Omron Sysmac Studio project Meca500_V9_3_3_Omron_EthernetIP_SquareMove_Demo_V1_1 (Sysmac Studio 1.53.0.64009, StandardProject)
(* Ajouter Calculate WRF function *)

# Controller NX1P2_1040DT1: NX1P2-1040DT1 version 1.16
Task PrimaryTask (priority 4, period or condition 2000): Meca500_E001

TYPE RobotControl : STRUCT
    Deactivate : BOOL;  (* offset 0.0 *)
    Activate : BOOL;  (* offset 0.1 *)
    Home : BOOL;  (* offset 0.2 *)
    ResetError : BOOL;  (* offset 0.3 *)
    EnableSimulation : BOOL;  (* offset 0.4 *)
    EnableRecoveryMode : BOOL;  (* offset 0.5 *)
END_STRUCT END_TYPE
TYPE Meca500 : STRUCT
    Outputs : Outputs;
    Inputs : Inputs;
    CommandsID : Meca500Cmd;
END_STRUCT END_TYPE
TYPE Inputs : STRUCT
    Status : Status;  (* offset 0.0 *)
    Motion : Motion;  (* offset 4.0 *)
    Joint_Set : Joint_Set;  (* offset 16.0 *)
    EndEffector_Pose : EndEffector_Pose;  (* offset 40.0 *)
    Configurations : Configurations;  (* offset 64.0 *)
    WRF : WRF;  (* offset 68.0 *)
    TRF : TRF;  (* offset 92.0 *)
    TimeStamp : TimeStamp;  (* offset 116.0 *)
    Reserved1 : SINT;  (* offset 128.0 *)
    Reserved2 : SINT;  (* offset 132.0 *)
    Reserved3 : SINT;  (* offset 136.0 *)
    DynamicData0 : DynamicData;  (* offset 140.0 *)
    DynamicData1 : DynamicData;  (* offset 168.0 *)
    DynamicData2 : DynamicData;  (* offset 196.0 *)
    DynamicData3 : DynamicData;  (* offset 224.0 *)
END_STRUCT END_TYPE
TYPE Status : STRUCT
    Busy : BOOL;
    Activated : BOOL;
    Homed : BOOL;
    SimActivated : BOOL;
    BrakesEngaged : BOOL;
    RecoveryMode : BOOL;
    EStop : BOOL;
    Error : UINT;
END_STRUCT END_TYPE
TYPE Motion : STRUCT
    CheckPoint : UDINT;  (* offset 0.0 *)
    MoveID : UINT;  (* offset 4.0 *)
    FifoSpace : UINT;  (* offset 6.0 *)
    Paused : BOOL;  (* offset 8.0 *)
    EOB : BOOL;  (* offset 8.1 *)
    EOM : BOOL;  (* offset 8.2 *)
    FifoCleared : BOOL;  (* offset 8.3 *)
    PStop2 : BOOL;  (* offset 8.4 *)
    ExcessiveTorque : BOOL;  (* offset 8.5 *)
    PStop2Resettable : BOOL;  (* offset 8.6 *)
    OfflineProgramID : UINT;  (* offset 10.0 *)
END_STRUCT END_TYPE
TYPE Joint_Set : STRUCT
    SubIndex001 : REAL;
    SubIndex002 : REAL;
    SubIndex003 : REAL;
    SubIndex004 : REAL;
    SubIndex005 : REAL;
    SubIndex006 : REAL;
END_STRUCT END_TYPE
TYPE EndEffector_Pose : STRUCT
    SubIndex001 : REAL;
    SubIndex002 : REAL;
    SubIndex003 : REAL;
    SubIndex004 : REAL;
    SubIndex005 : REAL;
    SubIndex006 : REAL;
END_STRUCT END_TYPE
TYPE Configurations : STRUCT
    Shoulder : SINT;  (* offset 0.0 *)
    Elbow : SINT;  (* offset 1.0 *)
    Wrist : SINT;  (* offset 2.0 *)
    Turn : SINT;  (* offset 3.0 *)
END_STRUCT END_TYPE
TYPE WRF : STRUCT
    SubIndex001 : REAL;
    SubIndex002 : REAL;
    SubIndex003 : REAL;
    SubIndex004 : REAL;
    SubIndex005 : REAL;
    SubIndex006 : REAL;
END_STRUCT END_TYPE
TYPE TRF : STRUCT
    SubIndex001 : REAL;
    SubIndex002 : REAL;
    SubIndex003 : REAL;
    SubIndex004 : REAL;
    SubIndex005 : REAL;
    SubIndex006 : REAL;
END_STRUCT END_TYPE
TYPE TimeStamp : STRUCT
    Seconds : UDINT;
    MicroSeconds : UDINT;
    DynamicDataCycles : UDINT;
END_STRUCT END_TYPE
TYPE DynamicData : STRUCT
    DynamicDataType : UDINT;
    DynamicDataValue0 : REAL;
    DynamicDataValue1 : REAL;
    DynamicDataValue2 : REAL;
    DynamicDataValue3 : REAL;
    DynamicDataValue4 : REAL;
    DynamicDataValue5 : REAL;
END_STRUCT END_TYPE
TYPE Outputs : STRUCT
    RobotControl : RobotControl;  (* offset 0.0 *)
    MotionControl : MotionControl;  (* offset 4.0 *)
    MotionCommand : MotionCommand;  (* offset 8.0 *)
    HostTime : UDINT;  (* offset 36.0 *)
    BrakesControlAllowed : BOOL;  (* offset 40.0 *)
    BrakesEngaged : BOOL;  (* offset 40.1 *)
    DynamicDataCfg0 : UDINT;  (* offset 44.0 *)
    DynamicDataCfg1 : UDINT;  (* offset 48.0 *)
    DynamicDataCfg2 : UDINT;  (* offset 52.0 *)
    DynamicDataCfg3 : UDINT;  (* offset 56.0 *)
END_STRUCT END_TYPE
TYPE MotionControl : STRUCT
    MoveID : UINT;  (* offset 0.0 *)
    Setpoint : BOOL;  (* offset 2.0 *)
    Pause : BOOL;  (* offset 2.1 *)
    CleaMove : BOOL;  (* offset 2.2 *)
    ResetPStop2 : BOOL;  (* offset 2.3 *)
END_STRUCT END_TYPE
TYPE MotionCommand : STRUCT
    MoveCommand : UDINT;  (* offset 0.0 *)
    MoveSubIndex001 : REAL;  (* offset 4.0 *)
    MoveSubIndex002 : REAL;  (* offset 8.0 *)
    MoveSubIndex003 : REAL;  (* offset 12.0 *)
    MoveSubIndex004 : REAL;  (* offset 16.0 *)
    MoveSubIndex005 : REAL;  (* offset 20.0 *)
    MoveSubIndex006 : REAL;  (* offset 24.0 *)
END_STRUCT END_TYPE
TYPE Meca500Cmd : (NoCmd := 0, MoveJoints := 1, MovePose := 2, MoveLin := 3, MoveLinRelTrf := 4, MoveLinRelWrf := 5, Delay := 6, SetBlending := 7, SetJointVel := 8, SetJointAcc := 9, SetCartAngVel := 10, SetCartLinVel := 11, SetCartAcc := 12, SetTrf := 13, SetWrf := 14, SetConf := 15, SetAutoConf := 16, SetCheckpoint := 17, Gripper := 18, SetGripperVel := 19, SetGripperForce := 20, MoveJointsVel := 21, MoveLinVelWrf := 22, MoveLinVelTrf := 23, SetVelTimeout := 24, SetConfTurn := 25, SetAutoConfTurn := 26, SetTorqueLimits := 27, SetTorquesLimitCfg := 28, MoveJointsRel := 29, SetValveState := 30, SetGripperRange := 31, MoveGripper := 32, SetJointVelLimit := 33, StartProgram := 100); END_TYPE

VAR_GLOBAL
    E001 : Meca500;  (* Robot Structure *)
    E001_Inputs : Inputs;  (* EthernetIp Inputs; network input *)
    E001_Outputs : Outputs;  (* EthernetIP Outputs; network output *)
END_VAR
VAR_GLOBAL CONSTANT
    Pi : REAL := 3.141592653589793238;
END_VAR

PROGRAM Meca500_E001
VAR
    Activate : BOOL;
    Deactivate : BOOL;
    Home : BOOL;
    ResetError : BOOL;
    Pause : BOOL;
    RecoveryMode : BOOL;
    StepSquareMove : INT;
    StartSequence : BOOL;
    SequenceActive : BOOL;
    SetCheckpoint1Buffered : BOOL;
    SetCartLinVel1Buffered : BOOL;
    MoveJoint1Buffered : BOOL;
    MovePose1Buffered : BOOL;
    MoveLin1Buffered : BOOL;
    Argument : ARRAY[0..5] OF real;
    SetCheckpoint1 : Meca500_SetCheckpoint;
    SetCartLinVel1 : Meca500_SetCartLinVel;
    MoveJoints1 : Meca500_MoveJoints;
    MovePose1 : Meca500_MovePose;
    MoveLin1 : Meca500_MoveLin;
END_VAR
VAR_EXTERNAL
    E001 : Meca500;
    E001_Inputs : Inputs;
    E001_Outputs : Outputs;
END_VAR
VAR
    _e1 : R_TRIG;
END_VAR

(* Section IOs: ladder, written here as Structured Text *)

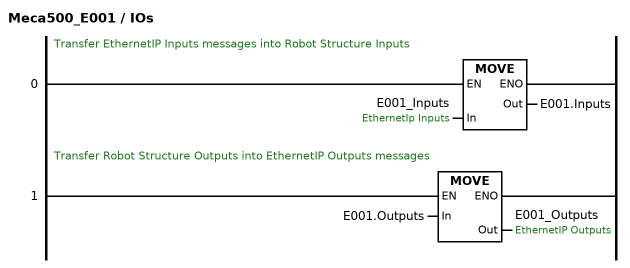
(* Rung 0: Transfer EthernetIP Inputs messages into Robot Structure Inputs *)
E001.Inputs := E001_Inputs;
(* Rung 1: Transfer Robot Structure Outputs into EthernetIP Outputs messages *)
E001_Outputs := E001.Outputs;

(* Section Robot_Control: ladder, written here as Structured Text *)

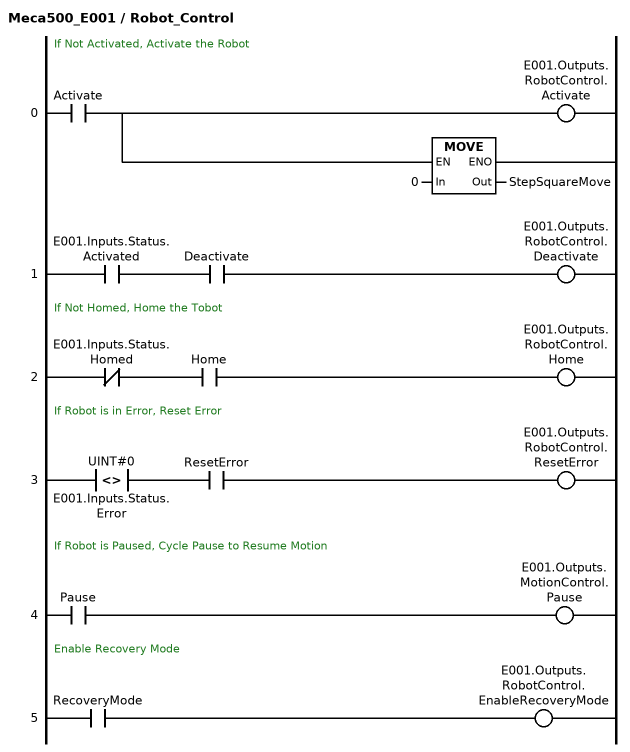
(* Rung 0: If Not Activated, Activate the Robot *)
E001.Outputs.RobotControl.Activate := Activate;
IF Activate THEN StepSquareMove := 0; END_IF;
(* Rung 1 *)
E001.Outputs.RobotControl.Deactivate := E001.Inputs.Status.Activated AND Deactivate;
(* Rung 2: If Not Homed, Home the Tobot *)
E001.Outputs.RobotControl.Home := NOT E001.Inputs.Status.Homed AND Home;
(* Rung 3: If Robot is in Error, Reset Error *)
E001.Outputs.RobotControl.ResetError := (UINT#0 <> E001.Inputs.Status.Error) AND ResetError;
(* Rung 4: If Robot is Paused, Cycle Pause to Resume Motion *)
E001.Outputs.MotionControl.Pause := Pause;
(* Rung 5: Enable Recovery Mode *)
E001.Outputs.RobotControl.EnableRecoveryMode := RecoveryMode;

(* Section Sequence: ladder, written here as Structured Text *)

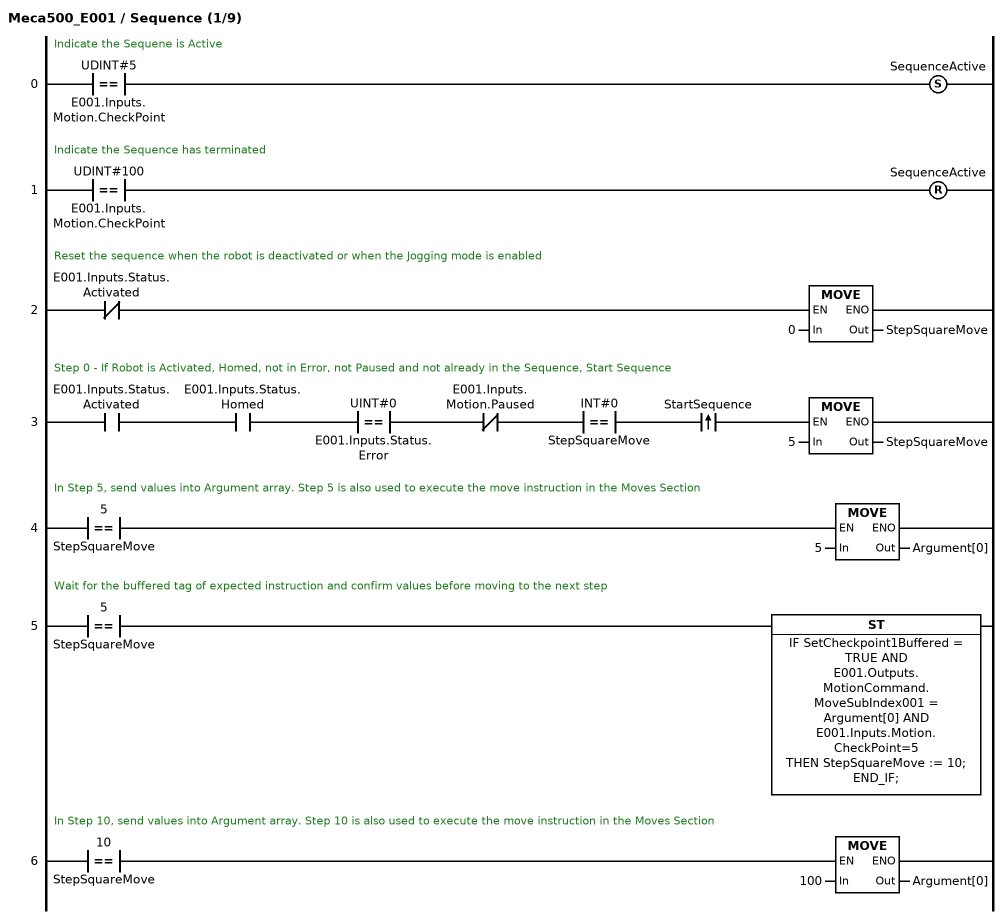
(* Rung 0: Indicate the Sequene is Active *)
IF UDINT#5 = E001.Inputs.Motion.CheckPoint THEN SequenceActive := TRUE; END_IF;
(* Rung 1: Indicate the Sequence has terminated *)
IF UDINT#100 = E001.Inputs.Motion.CheckPoint THEN SequenceActive := FALSE; END_IF;
(* Rung 2: Reset the sequence when the robot is deactivated or when the Jogging mode is enabled *)
IF NOT E001.Inputs.Status.Activated THEN StepSquareMove := 0; END_IF;
(* Rung 3: Step 0 - If Robot is Activated, Homed, not in Error, not Paused and not already in the Sequence, Start Sequence *)
_e1(CLK := StartSequence);
IF E001.Inputs.Status.Activated AND E001.Inputs.Status.Homed AND (UINT#0 = E001.Inputs.Status.Error) AND NOT E001.Inputs.Motion.Paused AND (INT#0 = StepSquareMove) AND _e1.Q THEN
    StepSquareMove := 5;
END_IF;
(* Rung 4: In Step 5, send values into Argument array. Step 5 is also used to execute the move instruction in the Moves Section *)
IF 5 = StepSquareMove THEN Argument[0] := 5; END_IF;
(* Rung 5: Wait for the buffered tag of expected instruction and confirm values before moving to the next step *)
IF 5 = StepSquareMove THEN
    IF SetCheckpoint1Buffered = TRUE AND
    	E001.Outputs.MotionCommand.MoveSubIndex001 = Argument[0] AND
    	E001.Inputs.Motion.CheckPoint=5
    	THEN StepSquareMove := 10;
    END_IF;
END_IF;
(* Rung 6: In Step 10, send values into Argument array. Step 10 is also used to execute the move instruction in the Moves Section *)
IF 10 = StepSquareMove THEN Argument[0] := 100; END_IF;

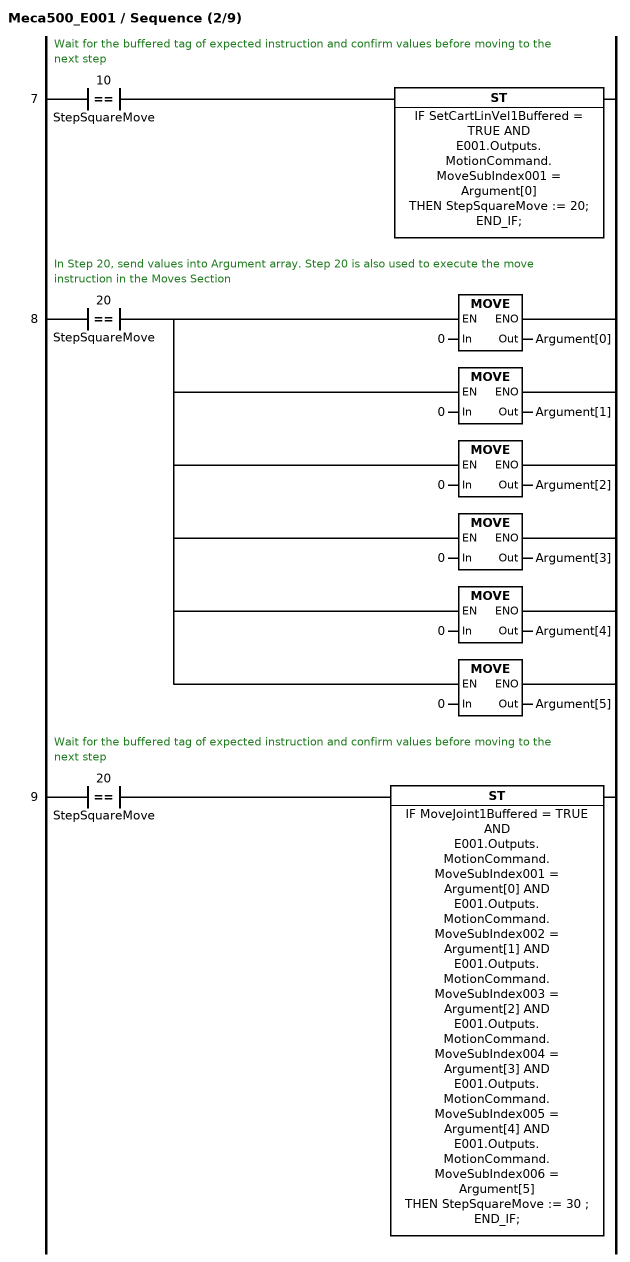
(* Rung 7: Wait for the buffered tag of expected instruction and confirm values before moving to the next step *)
IF 10 = StepSquareMove THEN
    IF SetCartLinVel1Buffered = TRUE AND
    	E001.Outputs.MotionCommand.MoveSubIndex001 = Argument[0]
    	THEN StepSquareMove := 20;
    END_IF;
END_IF;
(* Rung 8: In Step 20, send values into Argument array. Step 20 is also used to execute the move instruction in the Moves Section *)
IF 20 = StepSquareMove THEN
    Argument[0] := 0;
    Argument[1] := 0;
    Argument[2] := 0;
    Argument[3] := 0;
    Argument[4] := 0;
    Argument[5] := 0;
END_IF;
(* Rung 9: Wait for the buffered tag of expected instruction and confirm values before moving to the next step *)
IF 20 = StepSquareMove THEN
    IF MoveJoint1Buffered = TRUE AND
    	E001.Outputs.MotionCommand.MoveSubIndex001 = Argument[0] AND
    	E001.Outputs.MotionCommand.MoveSubIndex002 = Argument[1] AND
    	E001.Outputs.MotionCommand.MoveSubIndex003 = Argument[2] AND
    	E001.Outputs.MotionCommand.MoveSubIndex004 = Argument[3] AND
    	E001.Outputs.MotionCommand.MoveSubIndex005 = Argument[4] AND
    	E001.Outputs.MotionCommand.MoveSubIndex006 = Argument[5] 
    	THEN StepSquareMove := 30 ;
    END_IF;
END_IF;

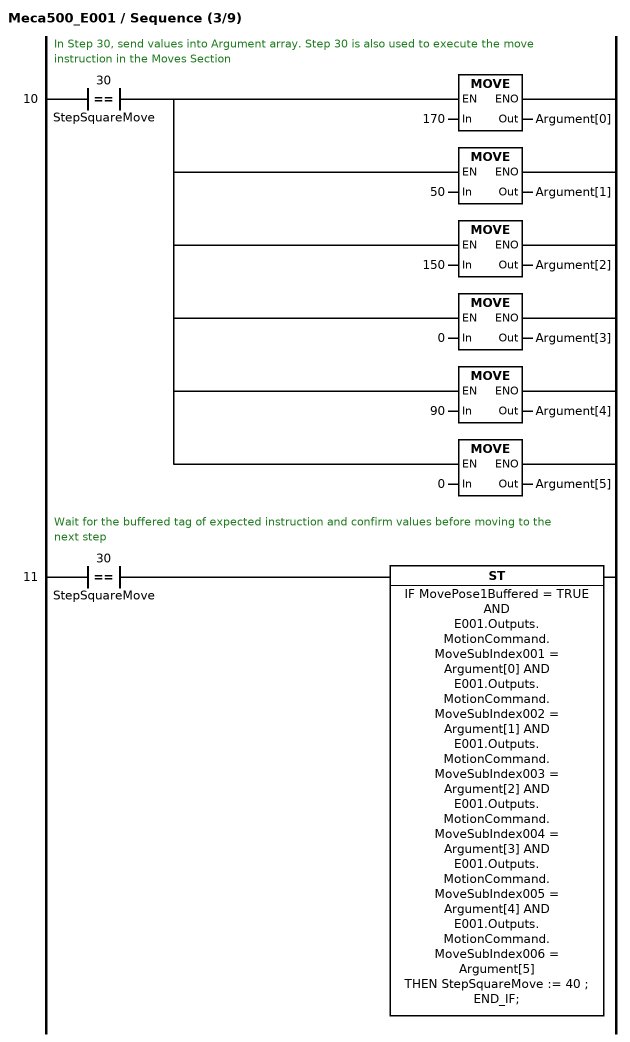
(* Rung 10: In Step 30, send values into Argument array. Step 30 is also used to execute the move instruction in the Moves Section *)
IF 30 = StepSquareMove THEN
    Argument[0] := 170;
    Argument[1] := 50;
    Argument[2] := 150;
    Argument[3] := 0;
    Argument[4] := 90;
    Argument[5] := 0;
END_IF;
(* Rung 11: Wait for the buffered tag of expected instruction and confirm values before moving to the next step *)
IF 30 = StepSquareMove THEN
    IF MovePose1Buffered = TRUE AND
    	E001.Outputs.MotionCommand.MoveSubIndex001 = Argument[0] AND
    	E001.Outputs.MotionCommand.MoveSubIndex002 = Argument[1] AND
    	E001.Outputs.MotionCommand.MoveSubIndex003 = Argument[2] AND
    	E001.Outputs.MotionCommand.MoveSubIndex004 = Argument[3] AND
    	E001.Outputs.MotionCommand.MoveSubIndex005 = Argument[4] AND
    	E001.Outputs.MotionCommand.MoveSubIndex006 = Argument[5] 
    	THEN StepSquareMove := 40 ;
    END_IF;
END_IF;

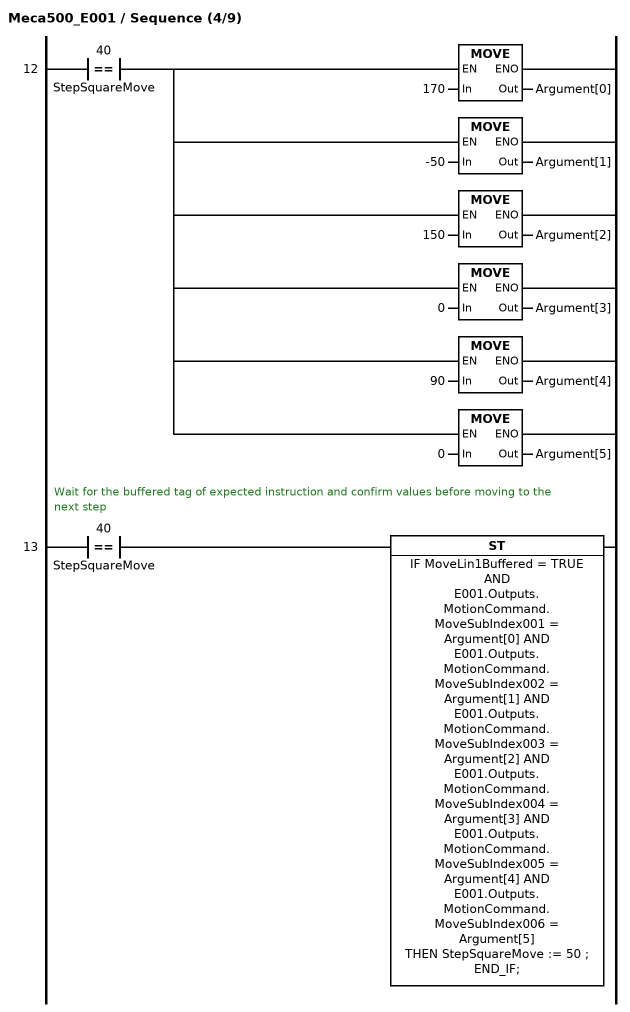
(* Rung 12 *)
IF 40 = StepSquareMove THEN
    Argument[0] := 170;
    Argument[1] := -50;
    Argument[2] := 150;
    Argument[3] := 0;
    Argument[4] := 90;
    Argument[5] := 0;
END_IF;
(* Rung 13: Wait for the buffered tag of expected instruction and confirm values before moving to the next step *)
IF 40 = StepSquareMove THEN
    IF MoveLin1Buffered = TRUE AND
    	E001.Outputs.MotionCommand.MoveSubIndex001 = Argument[0] AND
    	E001.Outputs.MotionCommand.MoveSubIndex002 = Argument[1] AND
    	E001.Outputs.MotionCommand.MoveSubIndex003 = Argument[2] AND
    	E001.Outputs.MotionCommand.MoveSubIndex004 = Argument[3] AND
    	E001.Outputs.MotionCommand.MoveSubIndex005 = Argument[4] AND
    	E001.Outputs.MotionCommand.MoveSubIndex006 = Argument[5] 
    	THEN StepSquareMove := 50 ;
    END_IF;
END_IF;

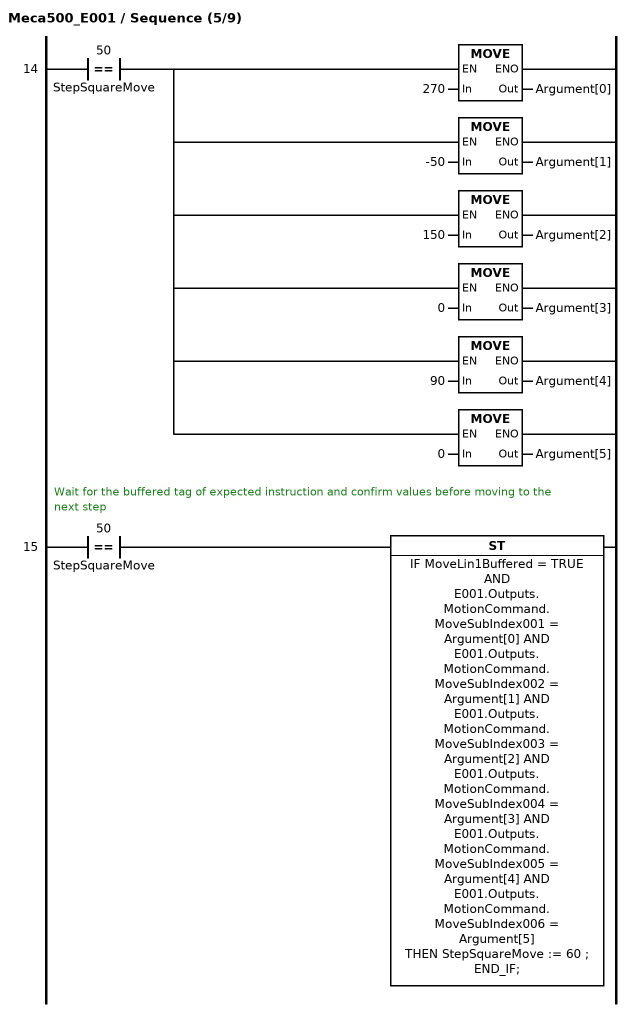
(* Rung 14 *)
IF 50 = StepSquareMove THEN
    Argument[0] := 270;
    Argument[1] := -50;
    Argument[2] := 150;
    Argument[3] := 0;
    Argument[4] := 90;
    Argument[5] := 0;
END_IF;
(* Rung 15: Wait for the buffered tag of expected instruction and confirm values before moving to the next step *)
IF 50 = StepSquareMove THEN
    IF MoveLin1Buffered = TRUE AND
    	E001.Outputs.MotionCommand.MoveSubIndex001 = Argument[0] AND
    	E001.Outputs.MotionCommand.MoveSubIndex002 = Argument[1] AND
    	E001.Outputs.MotionCommand.MoveSubIndex003 = Argument[2] AND
    	E001.Outputs.MotionCommand.MoveSubIndex004 = Argument[3] AND
    	E001.Outputs.MotionCommand.MoveSubIndex005 = Argument[4] AND
    	E001.Outputs.MotionCommand.MoveSubIndex006 = Argument[5] 
    	THEN StepSquareMove := 60 ;
    END_IF;
END_IF;

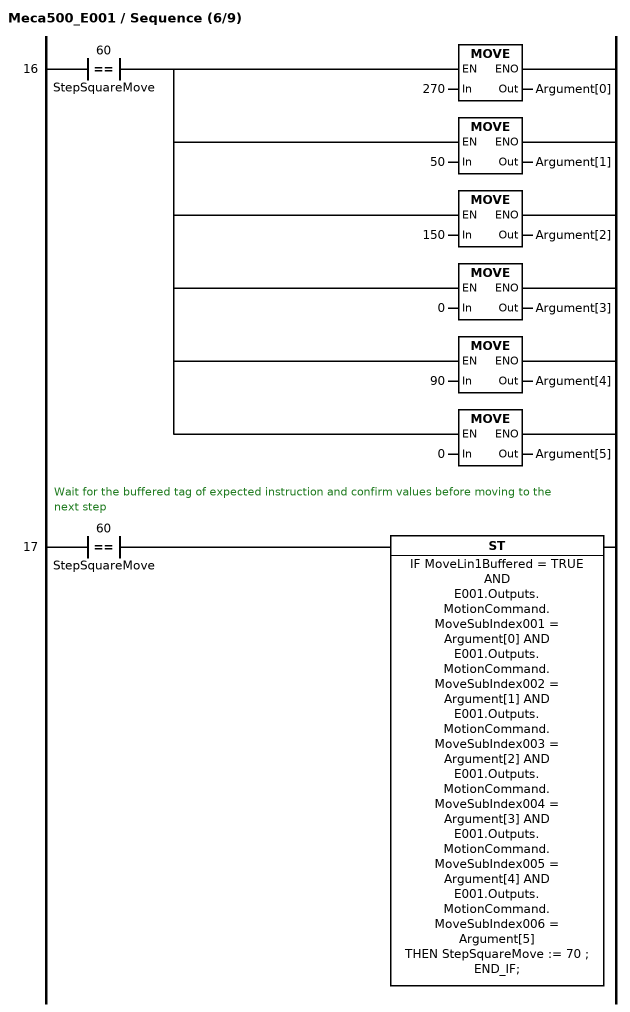
(* Rung 16 *)
IF 60 = StepSquareMove THEN
    Argument[0] := 270;
    Argument[1] := 50;
    Argument[2] := 150;
    Argument[3] := 0;
    Argument[4] := 90;
    Argument[5] := 0;
END_IF;
(* Rung 17: Wait for the buffered tag of expected instruction and confirm values before moving to the next step *)
IF 60 = StepSquareMove THEN
    IF MoveLin1Buffered = TRUE AND
    	E001.Outputs.MotionCommand.MoveSubIndex001 = Argument[0] AND
    	E001.Outputs.MotionCommand.MoveSubIndex002 = Argument[1] AND
    	E001.Outputs.MotionCommand.MoveSubIndex003 = Argument[2] AND
    	E001.Outputs.MotionCommand.MoveSubIndex004 = Argument[3] AND
    	E001.Outputs.MotionCommand.MoveSubIndex005 = Argument[4] AND
    	E001.Outputs.MotionCommand.MoveSubIndex006 = Argument[5] 
    	THEN StepSquareMove := 70 ;
    END_IF;
END_IF;

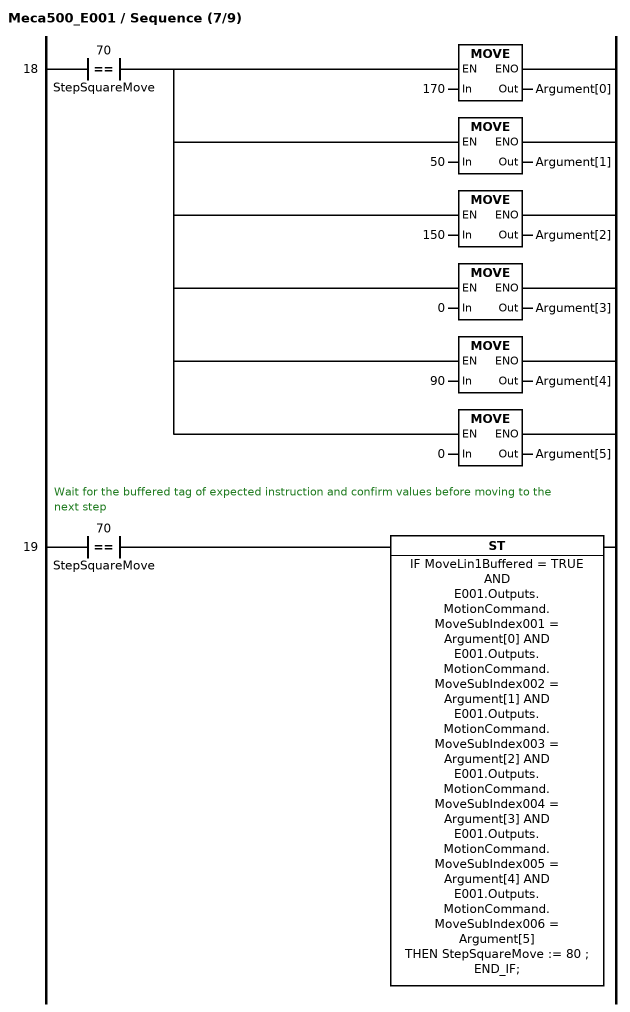
(* Rung 18 *)
IF 70 = StepSquareMove THEN
    Argument[0] := 170;
    Argument[1] := 50;
    Argument[2] := 150;
    Argument[3] := 0;
    Argument[4] := 90;
    Argument[5] := 0;
END_IF;
(* Rung 19: Wait for the buffered tag of expected instruction and confirm values before moving to the next step *)
IF 70 = StepSquareMove THEN
    IF MoveLin1Buffered = TRUE AND
    	E001.Outputs.MotionCommand.MoveSubIndex001 = Argument[0] AND
    	E001.Outputs.MotionCommand.MoveSubIndex002 = Argument[1] AND
    	E001.Outputs.MotionCommand.MoveSubIndex003 = Argument[2] AND
    	E001.Outputs.MotionCommand.MoveSubIndex004 = Argument[3] AND
    	E001.Outputs.MotionCommand.MoveSubIndex005 = Argument[4] AND
    	E001.Outputs.MotionCommand.MoveSubIndex006 = Argument[5] 
    	THEN StepSquareMove := 80 ;
    END_IF;
END_IF;

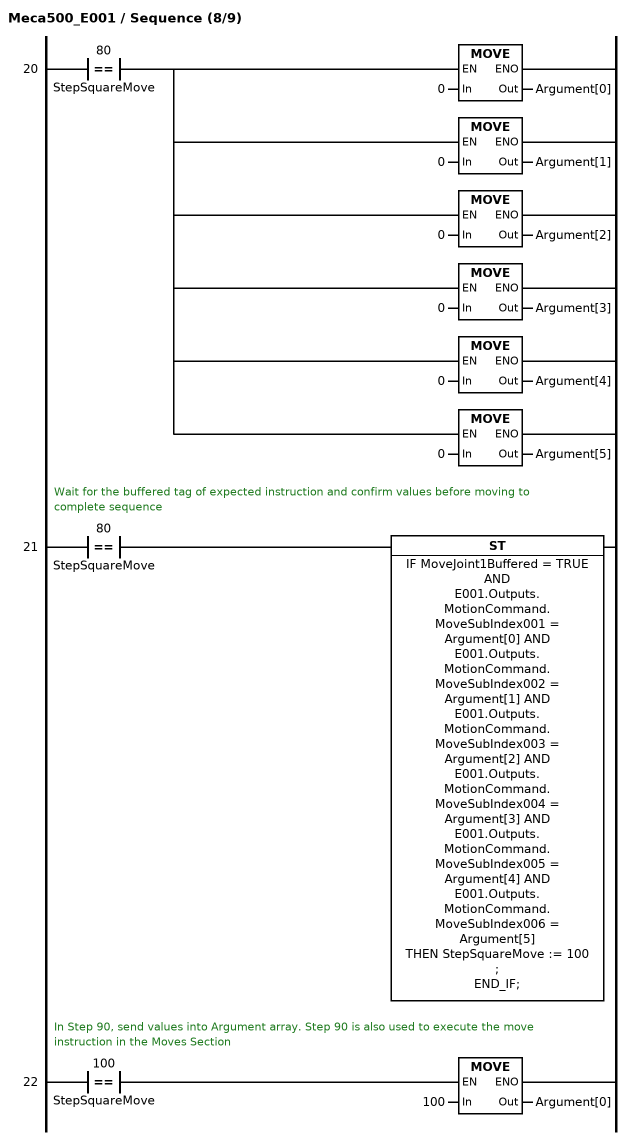
(* Rung 20 *)
IF 80 = StepSquareMove THEN
    Argument[0] := 0;
    Argument[1] := 0;
    Argument[2] := 0;
    Argument[3] := 0;
    Argument[4] := 0;
    Argument[5] := 0;
END_IF;
(* Rung 21: Wait for the buffered tag of expected instruction and confirm values before moving to complete sequence *)
IF 80 = StepSquareMove THEN
    IF MoveJoint1Buffered = TRUE AND
    	E001.Outputs.MotionCommand.MoveSubIndex001 = Argument[0] AND
    	E001.Outputs.MotionCommand.MoveSubIndex002 = Argument[1] AND
    	E001.Outputs.MotionCommand.MoveSubIndex003 = Argument[2] AND
    	E001.Outputs.MotionCommand.MoveSubIndex004 = Argument[3] AND
    	E001.Outputs.MotionCommand.MoveSubIndex005 = Argument[4] AND
    	E001.Outputs.MotionCommand.MoveSubIndex006 = Argument[5] 
    	THEN StepSquareMove := 100 ;
    END_IF;
END_IF;
(* Rung 22: In Step 90, send values into Argument array. Step 90 is also used to execute the move instruction in the Moves Section *)
IF 100 = StepSquareMove THEN Argument[0] := 100; END_IF;

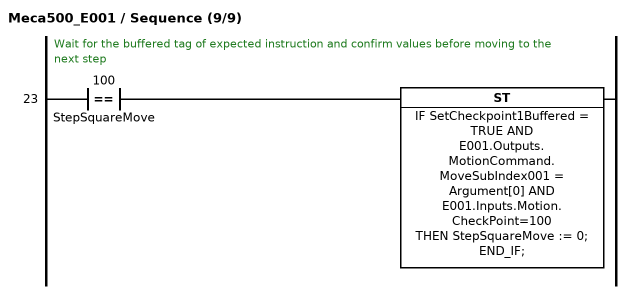
(* Rung 23: Wait for the buffered tag of expected instruction and confirm values before moving to the next step *)
IF 100 = StepSquareMove THEN
    IF SetCheckpoint1Buffered = TRUE AND
    	E001.Outputs.MotionCommand.MoveSubIndex001 = Argument[0] AND
    	E001.Inputs.Motion.CheckPoint=100
    	THEN StepSquareMove := 0;
    END_IF;
END_IF;

(* Section Instructions: ladder, written here as Structured Text *)

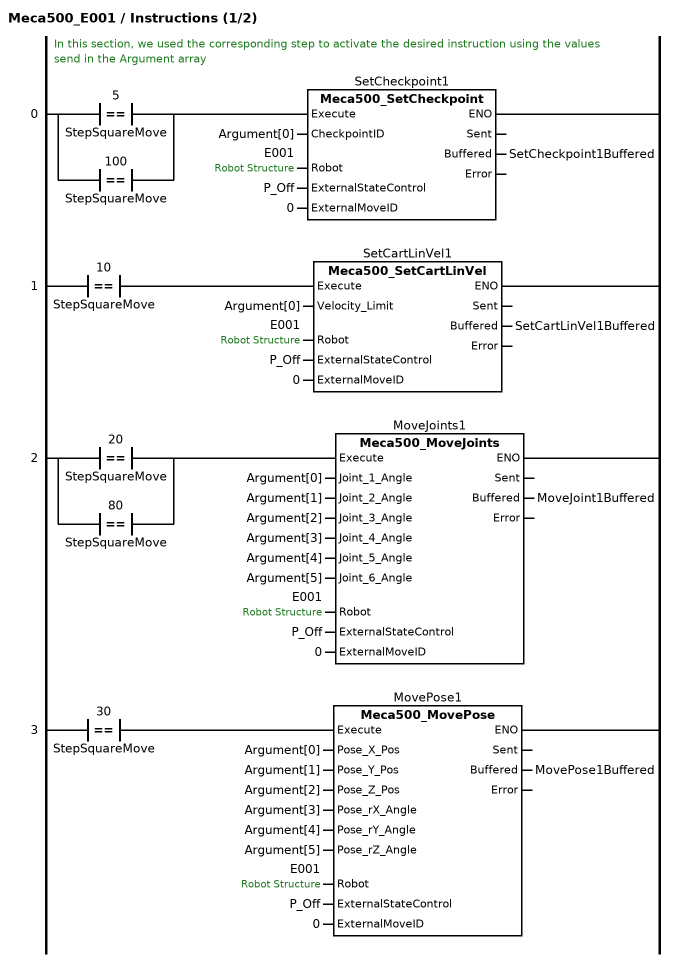
(* Rung 0: In this section, we used the corresponding step to activate the desired instruction using the values send in the Argument array *)
SetCheckpoint1(Execute := (5 = StepSquareMove) OR (100 = StepSquareMove), CheckpointID := Argument[0], Robot := E001, ExternalStateControl := P_Off, ExternalMoveID := 0, Buffered => SetCheckpoint1Buffered);
(* Rung 1 *)
SetCartLinVel1(Execute := 10 = StepSquareMove, Velocity_Limit := Argument[0], Robot := E001, ExternalStateControl := P_Off, ExternalMoveID := 0, Buffered => SetCartLinVel1Buffered);
(* Rung 2 *)
MoveJoints1(Execute := (20 = StepSquareMove) OR (80 = StepSquareMove), Joint_1_Angle := Argument[0], Joint_2_Angle := Argument[1], Joint_3_Angle := Argument[2], Joint_4_Angle := Argument[3], Joint_5_Angle := Argument[4], Joint_6_Angle := Argument[5], Robot := E001, ExternalStateControl := P_Off, ExternalMoveID := 0, Buffered => MoveJoint1Buffered);
(* Rung 3 *)
MovePose1(Execute := 30 = StepSquareMove, Pose_X_Pos := Argument[0], Pose_Y_Pos := Argument[1], Pose_Z_Pos := Argument[2], Pose_rX_Angle := Argument[3], Pose_rY_Angle := Argument[4], Pose_rZ_Angle := Argument[5], Robot := E001, ExternalStateControl := P_Off, ExternalMoveID := 0, Buffered => MovePose1Buffered);

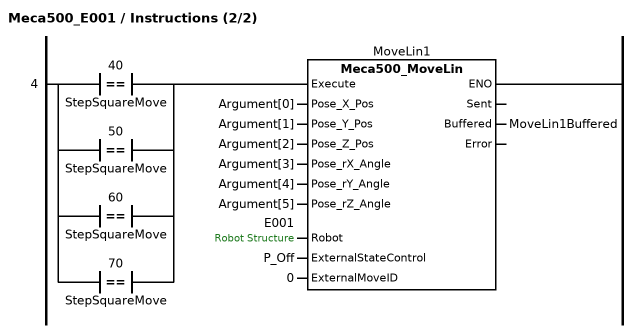
(* Rung 4 *)
MoveLin1(Execute := (40 = StepSquareMove) OR (50 = StepSquareMove) OR (60 = StepSquareMove) OR (70 = StepSquareMove), Pose_X_Pos := Argument[0], Pose_Y_Pos := Argument[1], Pose_Z_Pos := Argument[2], Pose_rX_Angle := Argument[3], Pose_rY_Angle := Argument[4], Pose_rZ_Angle := Argument[5], Robot := E001, ExternalStateControl := P_Off, ExternalMoveID := 0, Buffered => MoveLin1Buffered);
END_PROGRAM

FUNCTION atan2 : lREAL
VAR_INPUT
    y : lREAL;
    x : lREAL;
END_VAR
VAR_EXTERNAL CONSTANT
    Pi : REAL;
END_VAR
IF x > 0 THEN
	Atan2:=ATAN(y/x);
ELSIF x<0 AND y>=0 THEN
	Atan2:=ATAN(y/x)+Pi;
ELSIF  x<0 AND y<0 THEN
	Atan2:=ATAN(y/x)-Pi;
ELSIF  x=0 AND y>0 THEN
	Atan2:=Pi/2;
ELSIF  x=0 AND y<0 THEN
	Atan2:=-Pi/2;
END_IF;
END_FUNCTION

FUNCTION_BLOCK Meca500_Delay
VAR
    Output_Params : array[1..6] of real;
    FirstScan : BOOL := False;
END_VAR
VAR_INPUT
    Execute : BOOL;
    Seconds : REAL;
END_VAR
VAR_OUTPUT
    Sent : BOOL;
    Buffered : BOOL;
    Error : BOOL;
END_VAR
VAR_IN_OUT
    Robot : Meca500;
END_VAR
VAR_INPUT
    ExternalStateControl : BOOL;
    ExternalMoveID : UINT;
END_VAR
IF Execute THEN	
	(*Collect Inputs and store them locally*)
	Output_Params[1]:=Seconds;
	Output_Params[2]:=0;
	Output_Params[3]:=0;
	Output_Params[4]:=0;
	Output_Params[5]:=0;
	Output_Params[6]:=0;


	(* If Values have change, Reinitialise Outputs*)

	IF FirstScan=0 OR 
		Robot.Outputs.MotionCommand.MoveSubIndex001 <> Output_Params[1] OR 
		Robot.Outputs.MotionCommand.MoveSubIndex002 <> Output_Params[2] OR 
		Robot.Outputs.MotionCommand.MoveSubIndex003 <> Output_Params[3] OR
		Robot.Outputs.MotionCommand.MoveSubIndex004 <> Output_Params[4] OR 
		Robot.Outputs.MotionCommand.MoveSubIndex005 <> Output_Params[5] OR 
		Robot.Outputs.MotionCommand.MoveSubIndex006 <> Output_Params[6] 
	THEN
		Buffered := FALSE;
		Sent := FALSE;
	END_IF;


	(*if not in legacy mode, Act Setpoint*)
	IF Robot.Outputs.MotionControl.MoveID <> 0 THEN
	    Robot.Outputs.MotionControl.SetPoint := TRUE;
	END_IF;

	(* To send _Move, send _Move ID *)
	IF NOT Buffered AND NOT Sent THEN
	    
	    Robot.Outputs.MotionCommand.MoveCommand	:= EnumToNum(Meca500Cmd#Delay);
	    Robot.Outputs.MotionCommand.MoveSubIndex001 := Output_Params[1];
		Robot.Outputs.MotionCommand.MoveSubIndex002 := Output_Params[2];
		Robot.Outputs.MotionCommand.MoveSubIndex003 := Output_Params[3];
		Robot.Outputs.MotionCommand.MoveSubIndex004 := Output_Params[4];
		Robot.Outputs.MotionCommand.MoveSubIndex005 := Output_Params[5];
		Robot.Outputs.MotionCommand.MoveSubIndex006 := Output_Params[6];
	    
	    IF ExternalStateControl THEN
	        IF ExternalMoveID <> 0 AND ExternalMoveID <> 32060 AND ExternalMoveID <> 32061 THEN
	            Robot.Outputs.MotionControl.MoveID := ExternalMoveID;
	            Sent := TRUE;
	        END_IF;
	        
	    ELSE (*Not External Control*)
	        IF Robot.Outputs.MotionControl.MoveID = 32060 THEN
	            Robot.Outputs.MotionControl.MoveID := 32061;
	        ELSIF Robot.Outputs.MotionControl.MoveID = 32061 THEN
	            Robot.Outputs.MotionControl.MoveID := 32060;
	        ELSIF Robot.Outputs.MotionControl.MoveID <> 32060 OR Robot.Outputs.MotionControl.MoveID <> 32061 THEN
	            Robot.Outputs.MotionControl.MoveID := 32060;
	        END_IF;
	        Sent := TRUE;
	    END_IF;
	END_IF;

	(* Check if command has been sent, if so, check if it was received *)
	IF Sent AND
	    Robot.Outputs.MotionCommand.MoveCommand = EnumToNum(Meca500Cmd#Delay) AND
	    Robot.Outputs.MotionCommand.MoveSubIndex001 = Output_Params[1] AND 
		Robot.Outputs.MotionCommand.MoveSubIndex002 = Output_Params[2] AND 
		Robot.Outputs.MotionCommand.MoveSubIndex003 = Output_Params[3] AND 
		Robot.Outputs.MotionCommand.MoveSubIndex004 = Output_Params[4] AND 
		Robot.Outputs.MotionCommand.MoveSubIndex005 = Output_Params[5] AND 
		Robot.Outputs.MotionCommand.MoveSubIndex006 = Output_Params[6] AND
		Robot.Inputs.Motion.MoveID = Robot.Outputs.MotionControl.MoveID 
	THEN
		 Buffered := TRUE;
	END_IF;


	(*If External _Move ID is equal to Internal, raise an error*)
	IF ExternalMoveID = 32060 OR ExternalMoveID = 32061 THEN
	    Error := TRUE;
	END_IF;

	FirstScan := TRUE;
ELSE
	FirstScan := False;
	Sent := FALSE;
	Buffered := FALSE;
END_IF;
END_FUNCTION_BLOCK

FUNCTION_BLOCK Meca500_Gripper
VAR
    Output_Params : array[1..6] of real;
    FirstScan : BOOL := False;
END_VAR
VAR_INPUT
    Execute : BOOL;
    Open : REAL;
END_VAR
VAR_OUTPUT
    Sent : BOOL;
    Buffered : BOOL;
    Error : BOOL;
END_VAR
VAR_IN_OUT
    Robot : Meca500;
END_VAR
VAR_INPUT
    ExternalStateControl : BOOL;
    ExternalMoveID : UINT;
END_VAR
IF Execute THEN	
	(*Collect Inputs and store them locally*)
	Output_Params[1]:=Open;
	Output_Params[2]:=0;
	Output_Params[3]:=0;
	Output_Params[4]:=0;
	Output_Params[5]:=0;
	Output_Params[6]:=0;


	(* If Values have change, Reinitialise Outputs*)

	IF FirstScan=0 OR 
		Robot.Outputs.MotionCommand.MoveSubIndex001 <> Output_Params[1] OR 
		Robot.Outputs.MotionCommand.MoveSubIndex002 <> Output_Params[2] OR 
		Robot.Outputs.MotionCommand.MoveSubIndex003 <> Output_Params[3] OR
		Robot.Outputs.MotionCommand.MoveSubIndex004 <> Output_Params[4] OR 
		Robot.Outputs.MotionCommand.MoveSubIndex005 <> Output_Params[5] OR 
		Robot.Outputs.MotionCommand.MoveSubIndex006 <> Output_Params[6] 
	THEN
		Buffered := FALSE;
		Sent := FALSE;
	END_IF;


	(*if not in legacy mode, Act Setpoint*)
	IF Robot.Outputs.MotionControl.MoveID <> 0 THEN
	    Robot.Outputs.MotionControl.SetPoint := TRUE;
	END_IF;

	(* To send _Move, send _Move ID *)
	IF NOT Buffered AND NOT Sent THEN
	    
	    Robot.Outputs.MotionCommand.MoveCommand	:= EnumToNum(Meca500Cmd#Gripper);
	    Robot.Outputs.MotionCommand.MoveSubIndex001 := Output_Params[1];
		Robot.Outputs.MotionCommand.MoveSubIndex002 := Output_Params[2];
		Robot.Outputs.MotionCommand.MoveSubIndex003 := Output_Params[3];
		Robot.Outputs.MotionCommand.MoveSubIndex004 := Output_Params[4];
		Robot.Outputs.MotionCommand.MoveSubIndex005 := Output_Params[5];
		Robot.Outputs.MotionCommand.MoveSubIndex006 := Output_Params[6];
	    
	    IF ExternalStateControl THEN
	        IF ExternalMoveID <> 0 AND ExternalMoveID <> 32180 AND ExternalMoveID <> 32181 THEN
	            Robot.Outputs.MotionControl.MoveID := ExternalMoveID;
	            Sent := TRUE;
	        END_IF;
	        
	    ELSE (*Not External Control*)
	        IF Robot.Outputs.MotionControl.MoveID = 32180 THEN
	            Robot.Outputs.MotionControl.MoveID := 32181;
	        ELSIF Robot.Outputs.MotionControl.MoveID = 32181 THEN
	            Robot.Outputs.MotionControl.MoveID := 32180;
	        ELSIF Robot.Outputs.MotionControl.MoveID <> 32180 OR Robot.Outputs.MotionControl.MoveID <> 32181 THEN
	            Robot.Outputs.MotionControl.MoveID := 32180;
	        END_IF;
	        Sent := TRUE;
	    END_IF;
	END_IF;

	(* Check if command has been sent, if so, check if it was received *)
	IF Sent AND
	    Robot.Outputs.MotionCommand.MoveCommand = EnumToNum(Meca500Cmd#Gripper) AND
	    Robot.Outputs.MotionCommand.MoveSubIndex001 = Output_Params[1] AND 
		Robot.Outputs.MotionCommand.MoveSubIndex002 = Output_Params[2] AND 
		Robot.Outputs.MotionCommand.MoveSubIndex003 = Output_Params[3] AND 
		Robot.Outputs.MotionCommand.MoveSubIndex004 = Output_Params[4] AND 
		Robot.Outputs.MotionCommand.MoveSubIndex005 = Output_Params[5] AND 
		Robot.Outputs.MotionCommand.MoveSubIndex006 = Output_Params[6] AND
		Robot.Inputs.Motion.MoveID = Robot.Outputs.MotionControl.MoveID 
	THEN
		 Buffered := TRUE;
	END_IF;


	(*If External _Move ID is equal to Internal, raise an error*)
	IF ExternalMoveID = 32180 OR ExternalMoveID = 32181 THEN
	    Error := TRUE;
	END_IF;

	FirstScan := TRUE;
ELSE
	FirstScan := False;
	Sent := FALSE;
	Buffered := FALSE;
END_IF;
END_FUNCTION_BLOCK

FUNCTION_BLOCK Meca500_MoveGripper
VAR
    Output_Params : array[1..6] of real;
    FirstScan : BOOL := False;
END_VAR
VAR_INPUT
    Execute : BOOL;
    mm : REAL;
END_VAR
VAR_OUTPUT
    Sent : BOOL;
    Buffered : BOOL;
    Error : BOOL;
END_VAR
VAR_IN_OUT
    Robot : Meca500;
END_VAR
VAR_INPUT
    ExternalStateControl : BOOL;
    ExternalMoveID : UINT;
END_VAR
IF Execute THEN	
	(*Collect Inputs and store them locally*)
	Output_Params[1]:=mm;
	Output_Params[2]:=0;
	Output_Params[3]:=0;
	Output_Params[4]:=0;
	Output_Params[5]:=0;
	Output_Params[6]:=0;


	(* If Values have change, Reinitialise Outputs*)

	IF FirstScan=0 OR 
		Robot.Outputs.MotionCommand.MoveSubIndex001 <> Output_Params[1] OR 
		Robot.Outputs.MotionCommand.MoveSubIndex002 <> Output_Params[2] OR 
		Robot.Outputs.MotionCommand.MoveSubIndex003 <> Output_Params[3] OR
		Robot.Outputs.MotionCommand.MoveSubIndex004 <> Output_Params[4] OR 
		Robot.Outputs.MotionCommand.MoveSubIndex005 <> Output_Params[5] OR 
		Robot.Outputs.MotionCommand.MoveSubIndex006 <> Output_Params[6] 
	THEN
		Buffered := FALSE;
		Sent := FALSE;
	END_IF;


	(*if not in legacy mode, Act Setpoint*)
	IF Robot.Outputs.MotionControl.MoveID <> 0 THEN
	    Robot.Outputs.MotionControl.SetPoint := TRUE;
	END_IF;

	(* To send _Move, send _Move ID *)
	IF NOT Buffered AND NOT Sent THEN
	    
	    Robot.Outputs.MotionCommand.MoveCommand	:= EnumToNum(Meca500Cmd#MoveGripper);
	    Robot.Outputs.MotionCommand.MoveSubIndex001 := Output_Params[1];
		Robot.Outputs.MotionCommand.MoveSubIndex002 := Output_Params[2];
		Robot.Outputs.MotionCommand.MoveSubIndex003 := Output_Params[3];
		Robot.Outputs.MotionCommand.MoveSubIndex004 := Output_Params[4];
		Robot.Outputs.MotionCommand.MoveSubIndex005 := Output_Params[5];
		Robot.Outputs.MotionCommand.MoveSubIndex006 := Output_Params[6];
	    
	    IF ExternalStateControl THEN
	        IF ExternalMoveID <> 0 AND ExternalMoveID <> 32320 AND ExternalMoveID <> 32321 THEN
	            Robot.Outputs.MotionControl.MoveID := ExternalMoveID;
	            Sent := TRUE;
	        END_IF;
	        
	    ELSE (*Not External Control*)
	        IF Robot.Outputs.MotionControl.MoveID = 32320 THEN
	            Robot.Outputs.MotionControl.MoveID := 32321;
	        ELSIF Robot.Outputs.MotionControl.MoveID = 32321 THEN
	            Robot.Outputs.MotionControl.MoveID := 32320;
	        ELSIF Robot.Outputs.MotionControl.MoveID <> 32320 OR Robot.Outputs.MotionControl.MoveID <> 32321 THEN
	            Robot.Outputs.MotionControl.MoveID := 32320;
	        END_IF;
	        Sent := TRUE;
	    END_IF;
	END_IF;

	(* Check if command has been sent, if so, check if it was received *)
	IF Sent AND
	    Robot.Outputs.MotionCommand.MoveCommand = EnumToNum(Meca500Cmd#MoveGripper) AND
	    Robot.Outputs.MotionCommand.MoveSubIndex001 = Output_Params[1] AND 
		Robot.Outputs.MotionCommand.MoveSubIndex002 = Output_Params[2] AND 
		Robot.Outputs.MotionCommand.MoveSubIndex003 = Output_Params[3] AND 
		Robot.Outputs.MotionCommand.MoveSubIndex004 = Output_Params[4] AND 
		Robot.Outputs.MotionCommand.MoveSubIndex005 = Output_Params[5] AND 
		Robot.Outputs.MotionCommand.MoveSubIndex006 = Output_Params[6] AND
		Robot.Inputs.Motion.MoveID = Robot.Outputs.MotionControl.MoveID 
	THEN
		 Buffered := TRUE;
	END_IF;


	(*If External _Move ID is equal to Internal, raise an error*)
	IF ExternalMoveID = 32320 OR ExternalMoveID = 32321 THEN
	    Error := TRUE;
	END_IF;

	FirstScan := TRUE;
ELSE
	FirstScan := False;
	Sent := FALSE;
	Buffered := FALSE;
END_IF;
END_FUNCTION_BLOCK

FUNCTION_BLOCK Meca500_MoveJoints
VAR
    Output_Params : array[1..6] of real;
    FirstScan : BOOL := False;
END_VAR
VAR_INPUT
    Execute : BOOL;
    Joint_1_Angle : REAL;
    Joint_2_Angle : REAL;
    Joint_3_Angle : REAL;
    Joint_4_Angle : REAL;
    Joint_5_Angle : REAL;
    Joint_6_Angle : REAL;
END_VAR
VAR_OUTPUT
    Sent : BOOL;
    Buffered : BOOL;
    Error : BOOL;
END_VAR
VAR_IN_OUT
    Robot : Meca500;
END_VAR
VAR_INPUT
    ExternalStateControl : BOOL;
    ExternalMoveID : UINT;
END_VAR
IF Execute THEN	
	(*Collect Inputs and store them locally*)
	Output_Params[1]:=Joint_1_Angle;
	Output_Params[2]:=Joint_2_Angle;
	Output_Params[3]:=Joint_3_Angle;
	Output_Params[4]:=Joint_4_Angle;
	Output_Params[5]:=Joint_5_Angle;
	Output_Params[6]:=Joint_6_Angle;


	(* If Values have change, Reinitialise Outputs*)

	IF FirstScan=0 OR 
		Robot.Outputs.MotionCommand.MoveSubIndex001 <> Output_Params[1] OR 
		Robot.Outputs.MotionCommand.MoveSubIndex002 <> Output_Params[2] OR 
		Robot.Outputs.MotionCommand.MoveSubIndex003 <> Output_Params[3] OR
		Robot.Outputs.MotionCommand.MoveSubIndex004 <> Output_Params[4] OR 
		Robot.Outputs.MotionCommand.MoveSubIndex005 <> Output_Params[5] OR 
		Robot.Outputs.MotionCommand.MoveSubIndex006 <> Output_Params[6] 
	THEN
		Buffered := FALSE;
		Sent := FALSE;
	END_IF;


	(*if not in legacy mode, Act Setpoint*)
	IF Robot.Outputs.MotionControl.MoveID <> 0 THEN
	    Robot.Outputs.MotionControl.SetPoint := TRUE;
	END_IF;

	(* To send _Move, send _Move ID *)
	IF NOT Buffered AND NOT Sent THEN
	    
	    Robot.Outputs.MotionCommand.MoveCommand	:= EnumToNum(Meca500Cmd#MoveJoints);
	    Robot.Outputs.MotionCommand.MoveSubIndex001 := Output_Params[1];
		Robot.Outputs.MotionCommand.MoveSubIndex002 := Output_Params[2];
		Robot.Outputs.MotionCommand.MoveSubIndex003 := Output_Params[3];
		Robot.Outputs.MotionCommand.MoveSubIndex004 := Output_Params[4];
		Robot.Outputs.MotionCommand.MoveSubIndex005 := Output_Params[5];
		Robot.Outputs.MotionCommand.MoveSubIndex006 := Output_Params[6];
	    
	    IF ExternalStateControl THEN
	        IF ExternalMoveID <> 0 AND ExternalMoveID <> 32010 AND ExternalMoveID <> 32011 THEN
	            Robot.Outputs.MotionControl.MoveID := ExternalMoveID;
	            Sent := TRUE;
	        END_IF;
	        
	    ELSE (*Not External Control*)
	        IF Robot.Outputs.MotionControl.MoveID = 32010 THEN
	            Robot.Outputs.MotionControl.MoveID := 32011;
	        ELSIF Robot.Outputs.MotionControl.MoveID = 32011 THEN
	            Robot.Outputs.MotionControl.MoveID := 32010;
	        ELSIF Robot.Outputs.MotionControl.MoveID <> 32010 OR Robot.Outputs.MotionControl.MoveID <> 32011 THEN
	            Robot.Outputs.MotionControl.MoveID := 32010;
	        END_IF;
	        Sent := TRUE;
	    END_IF;
	END_IF;

	(* Check if command has been sent, if so, check if it was received *)
	IF Sent AND
	    Robot.Outputs.MotionCommand.MoveCommand = EnumToNum(Meca500Cmd#MoveJoints) AND
	    Robot.Outputs.MotionCommand.MoveSubIndex001 = Output_Params[1] AND 
		Robot.Outputs.MotionCommand.MoveSubIndex002 = Output_Params[2] AND 
		Robot.Outputs.MotionCommand.MoveSubIndex003 = Output_Params[3] AND 
		Robot.Outputs.MotionCommand.MoveSubIndex004 = Output_Params[4] AND 
		Robot.Outputs.MotionCommand.MoveSubIndex005 = Output_Params[5] AND 
		Robot.Outputs.MotionCommand.MoveSubIndex006 = Output_Params[6] AND
		Robot.Inputs.Motion.MoveID = Robot.Outputs.MotionControl.MoveID 
	THEN
		 Buffered := TRUE;
	END_IF;


	(*If External _Move ID is equal to Internal, raise an error*)
	IF ExternalMoveID = 32010 OR ExternalMoveID = 32011 THEN
	    Error := TRUE;
	END_IF;

	FirstScan := TRUE;
ELSE
	FirstScan := False;
	Sent := FALSE;
	Buffered := FALSE;
END_IF;
END_FUNCTION_BLOCK

FUNCTION_BLOCK Meca500_MoveJointsRel
VAR
    Output_Params : array[1..6] of real;
    FirstScan : BOOL := False;
END_VAR
VAR_INPUT
    Execute : BOOL;
    Joint_1_Angle : REAL;
    Joint_2_Angle : REAL;
    Joint_3_Angle : REAL;
    Joint_4_Angle : REAL;
    Joint_5_Angle : REAL;
    Joint_6_Angle : REAL;
END_VAR
VAR_OUTPUT
    Sent : BOOL;
    Buffered : BOOL;
    Error : BOOL;
END_VAR
VAR_IN_OUT
    Robot : Meca500;
END_VAR
VAR_INPUT
    ExternalStateControl : BOOL;
    ExternalMoveID : UINT;
END_VAR
IF Execute THEN	
	(*Collect Inputs and store them locally*)
	Output_Params[1]:=Joint_1_Angle;
	Output_Params[2]:=Joint_2_Angle;
	Output_Params[3]:=Joint_3_Angle;
	Output_Params[4]:=Joint_4_Angle;
	Output_Params[5]:=Joint_5_Angle;
	Output_Params[6]:=Joint_6_Angle;


	(* If Values have change, Reinitialise Outputs*)

	IF FirstScan=0 OR 
		Robot.Outputs.MotionCommand.MoveSubIndex001 <> Output_Params[1] OR 
		Robot.Outputs.MotionCommand.MoveSubIndex002 <> Output_Params[2] OR 
		Robot.Outputs.MotionCommand.MoveSubIndex003 <> Output_Params[3] OR
		Robot.Outputs.MotionCommand.MoveSubIndex004 <> Output_Params[4] OR 
		Robot.Outputs.MotionCommand.MoveSubIndex005 <> Output_Params[5] OR 
		Robot.Outputs.MotionCommand.MoveSubIndex006 <> Output_Params[6] 
	THEN
		Buffered := FALSE;
		Sent := FALSE;
	END_IF;


	(*if not in legacy mode, Act Setpoint*)
	IF Robot.Outputs.MotionControl.MoveID <> 0 THEN
	    Robot.Outputs.MotionControl.SetPoint := TRUE;
	END_IF;

	(* To send _Move, send _Move ID *)
	IF NOT Buffered AND NOT Sent THEN
	    
	    Robot.Outputs.MotionCommand.MoveCommand	:= EnumToNum(Meca500Cmd#MoveJointsRel);
	    Robot.Outputs.MotionCommand.MoveSubIndex001 := Output_Params[1];
		Robot.Outputs.MotionCommand.MoveSubIndex002 := Output_Params[2];
		Robot.Outputs.MotionCommand.MoveSubIndex003 := Output_Params[3];
		Robot.Outputs.MotionCommand.MoveSubIndex004 := Output_Params[4];
		Robot.Outputs.MotionCommand.MoveSubIndex005 := Output_Params[5];
		Robot.Outputs.MotionCommand.MoveSubIndex006 := Output_Params[6];
	    
	    IF ExternalStateControl THEN
	        IF ExternalMoveID <> 0 AND ExternalMoveID <> 32290 AND ExternalMoveID <> 32291 THEN
	            Robot.Outputs.MotionControl.MoveID := ExternalMoveID;
	            Sent := TRUE;
	        END_IF;
	        
	    ELSE (*Not External Control*)
	        IF Robot.Outputs.MotionControl.MoveID = 32290 THEN
	            Robot.Outputs.MotionControl.MoveID := 32291;
	        ELSIF Robot.Outputs.MotionControl.MoveID = 32291 THEN
	            Robot.Outputs.MotionControl.MoveID := 32290;
	        ELSIF Robot.Outputs.MotionControl.MoveID <> 32290 OR Robot.Outputs.MotionControl.MoveID <> 32291 THEN
	            Robot.Outputs.MotionControl.MoveID := 32290;
	        END_IF;
	        Sent := TRUE;
	    END_IF;
	END_IF;

	(* Check if command has been sent, if so, check if it was received *)
	IF Sent AND
	    Robot.Outputs.MotionCommand.MoveCommand = EnumToNum(Meca500Cmd#MoveJointsRel) AND
	    Robot.Outputs.MotionCommand.MoveSubIndex001 = Output_Params[1] AND 
		Robot.Outputs.MotionCommand.MoveSubIndex002 = Output_Params[2] AND 
		Robot.Outputs.MotionCommand.MoveSubIndex003 = Output_Params[3] AND 
		Robot.Outputs.MotionCommand.MoveSubIndex004 = Output_Params[4] AND 
		Robot.Outputs.MotionCommand.MoveSubIndex005 = Output_Params[5] AND 
		Robot.Outputs.MotionCommand.MoveSubIndex006 = Output_Params[6] AND
		Robot.Inputs.Motion.MoveID = Robot.Outputs.MotionControl.MoveID 
	THEN
		 Buffered := TRUE;
	END_IF;


	(*If External _Move ID is equal to Internal, raise an error*)
	IF ExternalMoveID = 32290 OR ExternalMoveID = 32291 THEN
	    Error := TRUE;
	END_IF;

	FirstScan := TRUE;
ELSE
	FirstScan := False;
	Sent := FALSE;
	Buffered := FALSE;
END_IF;
END_FUNCTION_BLOCK

FUNCTION_BLOCK Meca500_MoveJointsVel
VAR
    Output_Params : array[1..6] of real;
    FirstScan : BOOL := False;
END_VAR
VAR_INPUT
    Execute : BOOL;
    Joint_1_Vel : REAL;
    Joint_2_Vel : REAL;
    Joint_3_Vel : REAL;
    Joint_4_Vel : REAL;
    Joint_5_Vel : REAL;
    Joint_6_Vel : REAL;
END_VAR
VAR_OUTPUT
    Sent : BOOL;
    Buffered : BOOL;
    Error : BOOL;
END_VAR
VAR_IN_OUT
    Robot : Meca500;
END_VAR
VAR_INPUT
    ExternalStateControl : BOOL;
    ExternalMoveID : UINT;
END_VAR
IF Execute THEN	
	(*Collect Inputs and store them locally*)
	Output_Params[1]:=Joint_1_Vel;
	Output_Params[2]:=Joint_2_Vel;
	Output_Params[3]:=Joint_3_Vel;
	Output_Params[4]:=Joint_4_Vel;
	Output_Params[5]:=Joint_5_Vel;
	Output_Params[6]:=Joint_6_Vel;


	(* If Values have change, Reinitialise Outputs*)

	IF FirstScan=0 OR 
		Robot.Outputs.MotionCommand.MoveSubIndex001 <> Output_Params[1] OR 
		Robot.Outputs.MotionCommand.MoveSubIndex002 <> Output_Params[2] OR 
		Robot.Outputs.MotionCommand.MoveSubIndex003 <> Output_Params[3] OR
		Robot.Outputs.MotionCommand.MoveSubIndex004 <> Output_Params[4] OR 
		Robot.Outputs.MotionCommand.MoveSubIndex005 <> Output_Params[5] OR 
		Robot.Outputs.MotionCommand.MoveSubIndex006 <> Output_Params[6] 
	THEN
		Buffered := FALSE;
		Sent := FALSE;
	END_IF;


	(*if not in legacy mode, Act Setpoint*)
	IF Robot.Outputs.MotionControl.MoveID <> 0 THEN
	    Robot.Outputs.MotionControl.SetPoint := TRUE;
	END_IF;

	(* To send _Move, send _Move ID *)
	IF NOT Buffered AND NOT Sent THEN
	    
	    Robot.Outputs.MotionCommand.MoveCommand	:= EnumToNum(Meca500Cmd#MoveJointsVel);
	    Robot.Outputs.MotionCommand.MoveSubIndex001 := Output_Params[1];
		Robot.Outputs.MotionCommand.MoveSubIndex002 := Output_Params[2];
		Robot.Outputs.MotionCommand.MoveSubIndex003 := Output_Params[3];
		Robot.Outputs.MotionCommand.MoveSubIndex004 := Output_Params[4];
		Robot.Outputs.MotionCommand.MoveSubIndex005 := Output_Params[5];
		Robot.Outputs.MotionCommand.MoveSubIndex006 := Output_Params[6];
	    
	    IF ExternalStateControl THEN
	        IF ExternalMoveID <> 0 AND ExternalMoveID <> 32210 AND ExternalMoveID <> 32211 THEN
	            Robot.Outputs.MotionControl.MoveID := ExternalMoveID;
	            Sent := TRUE;
	        END_IF;
	        
	    ELSE (*Not External Control*)
	        IF Robot.Outputs.MotionControl.MoveID = 32210 THEN
	            Robot.Outputs.MotionControl.MoveID := 32211;
	        ELSIF Robot.Outputs.MotionControl.MoveID = 32211 THEN
	            Robot.Outputs.MotionControl.MoveID := 32210;
	        ELSIF Robot.Outputs.MotionControl.MoveID <> 32210 OR Robot.Outputs.MotionControl.MoveID <> 32211 THEN
	            Robot.Outputs.MotionControl.MoveID := 32210;
	        END_IF;
	        Sent := TRUE;
	    END_IF;
	END_IF;

	(* Check if command has been sent, if so, check if it was received *)
	IF Sent AND
	    Robot.Outputs.MotionCommand.MoveCommand = EnumToNum(Meca500Cmd#MoveJointsVel) AND
	    Robot.Outputs.MotionCommand.MoveSubIndex001 = Output_Params[1] AND 
		Robot.Outputs.MotionCommand.MoveSubIndex002 = Output_Params[2] AND 
		Robot.Outputs.MotionCommand.MoveSubIndex003 = Output_Params[3] AND 
		Robot.Outputs.MotionCommand.MoveSubIndex004 = Output_Params[4] AND 
		Robot.Outputs.MotionCommand.MoveSubIndex005 = Output_Params[5] AND 
		Robot.Outputs.MotionCommand.MoveSubIndex006 = Output_Params[6] AND
		Robot.Inputs.Motion.MoveID = Robot.Outputs.MotionControl.MoveID 
	THEN
		 Buffered := TRUE;
	END_IF;


	(*If External _Move ID is equal to Internal, raise an error*)
	IF ExternalMoveID = 32210 OR ExternalMoveID = 32211 THEN
	    Error := TRUE;
	END_IF;

	FirstScan := TRUE;
ELSE
	FirstScan := False;
	Sent := FALSE;
	Buffered := FALSE;
END_IF;
END_FUNCTION_BLOCK

FUNCTION_BLOCK Meca500_MoveLin
VAR
    Output_Params : array[1..6] of real;
    FirstScan : BOOL := False;
END_VAR
VAR_INPUT
    Execute : BOOL;
    Pose_X_Pos : REAL;
    Pose_Y_Pos : REAL;
    Pose_Z_Pos : REAL;
    Pose_rX_Angle : REAL;
    Pose_rY_Angle : REAL;
    Pose_rZ_Angle : REAL;
END_VAR
VAR_OUTPUT
    Sent : BOOL;
    Buffered : BOOL;
    Error : BOOL;
END_VAR
VAR_IN_OUT
    Robot : Meca500;
END_VAR
VAR_INPUT
    ExternalStateControl : BOOL;
    ExternalMoveID : UINT;
END_VAR
IF Execute THEN	
	(*Collect Inputs and store them locally*)
	Output_Params[1]:=Pose_X_Pos;
	Output_Params[2]:=Pose_Y_Pos;
	Output_Params[3]:=Pose_Z_Pos;
	Output_Params[4]:=Pose_rX_Angle;
	Output_Params[5]:=Pose_rY_Angle;
	Output_Params[6]:=Pose_rZ_Angle;

	(* If Values have change, Reinitialise Outputs*)

	IF FirstScan=0 OR 
		Robot.Outputs.MotionCommand.MoveSubIndex001 <> Output_Params[1] OR 
		Robot.Outputs.MotionCommand.MoveSubIndex002 <> Output_Params[2] OR 
		Robot.Outputs.MotionCommand.MoveSubIndex003 <> Output_Params[3] OR
		Robot.Outputs.MotionCommand.MoveSubIndex004 <> Output_Params[4] OR 
		Robot.Outputs.MotionCommand.MoveSubIndex005 <> Output_Params[5] OR 
		Robot.Outputs.MotionCommand.MoveSubIndex006 <> Output_Params[6] 
	THEN
		Buffered := FALSE;
		Sent := FALSE;
	END_IF;


	(*if not in legacy mode, Act Setpoint*)
	IF Robot.Outputs.MotionControl.MoveID <> 0 THEN
	    Robot.Outputs.MotionControl.SetPoint := TRUE;
	END_IF;

	(* To send _Move, send _Move ID *)
	IF NOT Buffered AND NOT Sent THEN
	    
	    Robot.Outputs.MotionCommand.MoveCommand	:= EnumToNum(Meca500Cmd#MoveLin);
	    Robot.Outputs.MotionCommand.MoveSubIndex001 := Output_Params[1];
		Robot.Outputs.MotionCommand.MoveSubIndex002 := Output_Params[2];
		Robot.Outputs.MotionCommand.MoveSubIndex003 := Output_Params[3];
		Robot.Outputs.MotionCommand.MoveSubIndex004 := Output_Params[4];
		Robot.Outputs.MotionCommand.MoveSubIndex005 := Output_Params[5];
		Robot.Outputs.MotionCommand.MoveSubIndex006 := Output_Params[6];
	    
	    IF ExternalStateControl THEN
	        IF ExternalMoveID <> 0 AND ExternalMoveID <> 32030 AND ExternalMoveID <> 32031 THEN
	            Robot.Outputs.MotionControl.MoveID := ExternalMoveID;
	            Sent := TRUE;
	        END_IF;
	        
	    ELSE (*Not External Control*)
	        IF Robot.Outputs.MotionControl.MoveID = 32030 THEN
	            Robot.Outputs.MotionControl.MoveID := 32031;
	        ELSIF Robot.Outputs.MotionControl.MoveID = 32031 THEN
	            Robot.Outputs.MotionControl.MoveID := 32030;
	        ELSIF Robot.Outputs.MotionControl.MoveID <> 32030 OR Robot.Outputs.MotionControl.MoveID <> 32031 THEN
	            Robot.Outputs.MotionControl.MoveID := 32030;
	        END_IF;
	        Sent := TRUE;
	    END_IF;
	END_IF;

	(* Check if command has been sent, if so, check if it was received *)
	IF Sent AND
	    Robot.Outputs.MotionCommand.MoveCommand = EnumToNum(Meca500Cmd#MoveLin) AND
	    Robot.Outputs.MotionCommand.MoveSubIndex001 = Output_Params[1] AND 
		Robot.Outputs.MotionCommand.MoveSubIndex002 = Output_Params[2] AND 
		Robot.Outputs.MotionCommand.MoveSubIndex003 = Output_Params[3] AND 
		Robot.Outputs.MotionCommand.MoveSubIndex004 = Output_Params[4] AND 
		Robot.Outputs.MotionCommand.MoveSubIndex005 = Output_Params[5] AND 
		Robot.Outputs.MotionCommand.MoveSubIndex006 = Output_Params[6] AND
		Robot.Inputs.Motion.MoveID = Robot.Outputs.MotionControl.MoveID 
	THEN
		 Buffered := TRUE;
	END_IF;


	(*If External _Move ID is equal to Internal, raise an error*)
	IF ExternalMoveID = 32030 OR ExternalMoveID = 32031 THEN
	    Error := TRUE;
	END_IF;

	FirstScan := TRUE;
ELSE
	FirstScan := False;
	Sent := FALSE;
	Buffered := FALSE;
END_IF;
END_FUNCTION_BLOCK

FUNCTION_BLOCK Meca500_MoveLinRelTRF
VAR
    Output_Params : array[1..6] of real;
    FirstScan : BOOL := False;
END_VAR
VAR_INPUT
    Execute : BOOL;
    Pose_X_Pos : REAL;
    Pose_Y_Pos : REAL;
    Pose_Z_Pos : REAL;
    Pose_rX_Angle : REAL;
    Pose_rY_Angle : REAL;
    Pose_rZ_Angle : REAL;
END_VAR
VAR_OUTPUT
    Sent : BOOL;
    Buffered : BOOL;
    Error : BOOL;
END_VAR
VAR_IN_OUT
    Robot : Meca500;
END_VAR
VAR_INPUT
    ExternalStateControl : BOOL;
    ExternalMoveID : UINT;
END_VAR
IF Execute THEN	
	(*Collect Inputs and store them locally*)
	Output_Params[1]:=Pose_X_Pos;
	Output_Params[2]:=Pose_Y_Pos;
	Output_Params[3]:=Pose_Z_Pos;
	Output_Params[4]:=Pose_rX_Angle;
	Output_Params[5]:=Pose_rY_Angle;
	Output_Params[6]:=Pose_rZ_Angle;

	(* If Values have change, Reinitialise Outputs*)

	IF FirstScan=0 OR 
		Robot.Outputs.MotionCommand.MoveSubIndex001 <> Output_Params[1] OR 
		Robot.Outputs.MotionCommand.MoveSubIndex002 <> Output_Params[2] OR 
		Robot.Outputs.MotionCommand.MoveSubIndex003 <> Output_Params[3] OR
		Robot.Outputs.MotionCommand.MoveSubIndex004 <> Output_Params[4] OR 
		Robot.Outputs.MotionCommand.MoveSubIndex005 <> Output_Params[5] OR 
		Robot.Outputs.MotionCommand.MoveSubIndex006 <> Output_Params[6] 
	THEN
		Buffered := FALSE;
		Sent := FALSE;
	END_IF;


	(*if not in legacy mode, Act Setpoint*)
	IF Robot.Outputs.MotionControl.MoveID <> 0 THEN
	    Robot.Outputs.MotionControl.SetPoint := TRUE;
	END_IF;

	(* To send _Move, send _Move ID *)
	IF NOT Buffered AND NOT Sent THEN
	    
	    Robot.Outputs.MotionCommand.MoveCommand	:= EnumToNum(Meca500Cmd#MoveLinRelTrf);
	    Robot.Outputs.MotionCommand.MoveSubIndex001 := Output_Params[1];
		Robot.Outputs.MotionCommand.MoveSubIndex002 := Output_Params[2];
		Robot.Outputs.MotionCommand.MoveSubIndex003 := Output_Params[3];
		Robot.Outputs.MotionCommand.MoveSubIndex004 := Output_Params[4];
		Robot.Outputs.MotionCommand.MoveSubIndex005 := Output_Params[5];
		Robot.Outputs.MotionCommand.MoveSubIndex006 := Output_Params[6];
	    
	    IF ExternalStateControl THEN
	        IF ExternalMoveID <> 0 AND ExternalMoveID <> 32040 AND ExternalMoveID <> 32041 THEN
	            Robot.Outputs.MotionControl.MoveID := ExternalMoveID;
	            Sent := TRUE;
	        END_IF;
	        
	    ELSE (*Not External Control*)
	        IF Robot.Outputs.MotionControl.MoveID = 32040 THEN
	            Robot.Outputs.MotionControl.MoveID := 32041;
	        ELSIF Robot.Outputs.MotionControl.MoveID = 32041 THEN
	            Robot.Outputs.MotionControl.MoveID := 32040;
	        ELSIF Robot.Outputs.MotionControl.MoveID <> 32040 OR Robot.Outputs.MotionControl.MoveID <> 32041 THEN
	            Robot.Outputs.MotionControl.MoveID := 32040;
	        END_IF;
	        Sent := TRUE;
	    END_IF;
	END_IF;

	(* Check if command has been sent, if so, check if it was received *)
	IF Sent AND
	    Robot.Outputs.MotionCommand.MoveCommand = EnumToNum(Meca500Cmd#MoveLinRelTrf) AND
	    Robot.Outputs.MotionCommand.MoveSubIndex001 = Output_Params[1] AND 
		Robot.Outputs.MotionCommand.MoveSubIndex002 = Output_Params[2] AND 
		Robot.Outputs.MotionCommand.MoveSubIndex003 = Output_Params[3] AND 
		Robot.Outputs.MotionCommand.MoveSubIndex004 = Output_Params[4] AND 
		Robot.Outputs.MotionCommand.MoveSubIndex005 = Output_Params[5] AND 
		Robot.Outputs.MotionCommand.MoveSubIndex006 = Output_Params[6] AND
		Robot.Inputs.Motion.MoveID = Robot.Outputs.MotionControl.MoveID 
	THEN
		 Buffered := TRUE;
	END_IF;


	(*If External _Move ID is equal to Internal, raise an error*)
	IF ExternalMoveID = 32040 OR ExternalMoveID = 32041 THEN
	    Error := TRUE;
	END_IF;

	FirstScan := TRUE;
ELSE
	FirstScan := False;
	Sent := FALSE;
	Buffered := FALSE;
END_IF;
END_FUNCTION_BLOCK

FUNCTION_BLOCK Meca500_MoveLinRelWRF
VAR
    Output_Params : array[1..6] of real;
    FirstScan : BOOL := False;
END_VAR
VAR_INPUT
    Execute : BOOL;
    Pose_X_Pos : REAL;
    Pose_Y_Pos : REAL;
    Pose_Z_Pos : REAL;
    Pose_rX_Angle : REAL;
    Pose_rY_Angle : REAL;
    Pose_rZ_Angle : REAL;
END_VAR
VAR_OUTPUT
    Sent : BOOL;
    Buffered : BOOL;
    Error : BOOL;
END_VAR
VAR_IN_OUT
    Robot : Meca500;
END_VAR
VAR_INPUT
    ExternalStateControl : BOOL;
    ExternalMoveID : UINT;
END_VAR
IF Execute THEN	
	(*Collect Inputs and store them locally*)
	Output_Params[1]:=Pose_X_Pos;
	Output_Params[2]:=Pose_Y_Pos;
	Output_Params[3]:=Pose_Z_Pos;
	Output_Params[4]:=Pose_rX_Angle;
	Output_Params[5]:=Pose_rY_Angle;
	Output_Params[6]:=Pose_rZ_Angle;

	(* If Values have change, Reinitialise Outputs*)

	IF FirstScan=0 OR 
		Robot.Outputs.MotionCommand.MoveSubIndex001 <> Output_Params[1] OR 
		Robot.Outputs.MotionCommand.MoveSubIndex002 <> Output_Params[2] OR 
		Robot.Outputs.MotionCommand.MoveSubIndex003 <> Output_Params[3] OR
		Robot.Outputs.MotionCommand.MoveSubIndex004 <> Output_Params[4] OR 
		Robot.Outputs.MotionCommand.MoveSubIndex005 <> Output_Params[5] OR 
		Robot.Outputs.MotionCommand.MoveSubIndex006 <> Output_Params[6] 
	THEN
		Buffered := FALSE;
		Sent := FALSE;
	END_IF;


	(*if not in legacy mode, Act Setpoint*)
	IF Robot.Outputs.MotionControl.MoveID <> 0 THEN
	    Robot.Outputs.MotionControl.SetPoint := TRUE;
	END_IF;

	(* To send _Move, send _Move ID *)
	IF NOT Buffered AND NOT Sent THEN
	    
	    Robot.Outputs.MotionCommand.MoveCommand	:= EnumToNum(Meca500Cmd#MoveLinRelWrf);
	    Robot.Outputs.MotionCommand.MoveSubIndex001 := Output_Params[1];
		Robot.Outputs.MotionCommand.MoveSubIndex002 := Output_Params[2];
		Robot.Outputs.MotionCommand.MoveSubIndex003 := Output_Params[3];
		Robot.Outputs.MotionCommand.MoveSubIndex004 := Output_Params[4];
		Robot.Outputs.MotionCommand.MoveSubIndex005 := Output_Params[5];
		Robot.Outputs.MotionCommand.MoveSubIndex006 := Output_Params[6];
	    
	    IF ExternalStateControl THEN
	        IF ExternalMoveID <> 0 AND ExternalMoveID <> 32050 AND ExternalMoveID <> 32051 THEN
	            Robot.Outputs.MotionControl.MoveID := ExternalMoveID;
	            Sent := TRUE;
	        END_IF;
	        
	    ELSE (*Not External Control*)
	        IF Robot.Outputs.MotionControl.MoveID = 32050 THEN
	            Robot.Outputs.MotionControl.MoveID := 32051;
	        ELSIF Robot.Outputs.MotionControl.MoveID = 32051 THEN
	            Robot.Outputs.MotionControl.MoveID := 32050;
	        ELSIF Robot.Outputs.MotionControl.MoveID <> 32050 OR Robot.Outputs.MotionControl.MoveID <> 32051 THEN
	            Robot.Outputs.MotionControl.MoveID := 32050;
	        END_IF;
	        Sent := TRUE;
	    END_IF;
	END_IF;

	(* Check if command has been sent, if so, check if it was received *)
	IF Sent AND
	    Robot.Outputs.MotionCommand.MoveCommand = EnumToNum(Meca500Cmd#MoveLinRelWrf) AND
	    Robot.Outputs.MotionCommand.MoveSubIndex001 = Output_Params[1] AND 
		Robot.Outputs.MotionCommand.MoveSubIndex002 = Output_Params[2] AND 
		Robot.Outputs.MotionCommand.MoveSubIndex003 = Output_Params[3] AND 
		Robot.Outputs.MotionCommand.MoveSubIndex004 = Output_Params[4] AND 
		Robot.Outputs.MotionCommand.MoveSubIndex005 = Output_Params[5] AND 
		Robot.Outputs.MotionCommand.MoveSubIndex006 = Output_Params[6] AND
		Robot.Inputs.Motion.MoveID = Robot.Outputs.MotionControl.MoveID 
	THEN
		 Buffered := TRUE;
	END_IF;


	(*If External _Move ID is equal to Internal, raise an error*)
	IF ExternalMoveID = 32050 OR ExternalMoveID = 32051 THEN
	    Error := TRUE;
	END_IF;

	FirstScan := TRUE;
ELSE
	FirstScan := False;
	Sent := FALSE;
	Buffered := FALSE;
END_IF;
END_FUNCTION_BLOCK

FUNCTION_BLOCK Meca500_MoveLinVelTRF
VAR
    Output_Params : array[1..6] of real;
    FirstScan : BOOL := False;
END_VAR
VAR_INPUT
    Execute : BOOL;
    X_Vel : REAL;
    Y_Vel : REAL;
    Z_Vel : REAL;
    rX_AngleVel : REAL;
    rY_AngleVel : REAL;
    rZ_AngleVel : REAL;
END_VAR
VAR_OUTPUT
    Sent : BOOL;
    Buffered : BOOL;
    Error : BOOL;
END_VAR
VAR_IN_OUT
    Robot : Meca500;
END_VAR
VAR_INPUT
    ExternalStateControl : BOOL;
    ExternalMoveID : UINT;
END_VAR
IF Execute THEN	
	(*Collect Inputs and store them locally*)
	Output_Params[1]:=X_Vel;
	Output_Params[2]:=Y_Vel;
	Output_Params[3]:=Z_Vel;
	Output_Params[4]:=rX_AngleVel;
	Output_Params[5]:=rY_AngleVel;
	Output_Params[6]:=rZ_AngleVel;

	(* If Values have change, Reinitialise Outputs*)

	IF FirstScan=0 OR 
		Robot.Outputs.MotionCommand.MoveSubIndex001 <> Output_Params[1] OR 
		Robot.Outputs.MotionCommand.MoveSubIndex002 <> Output_Params[2] OR 
		Robot.Outputs.MotionCommand.MoveSubIndex003 <> Output_Params[3] OR
		Robot.Outputs.MotionCommand.MoveSubIndex004 <> Output_Params[4] OR 
		Robot.Outputs.MotionCommand.MoveSubIndex005 <> Output_Params[5] OR 
		Robot.Outputs.MotionCommand.MoveSubIndex006 <> Output_Params[6] 
	THEN
		Buffered := FALSE;
		Sent := FALSE;
	END_IF;


	(*if not in legacy mode, Act Setpoint*)
	IF Robot.Outputs.MotionControl.MoveID <> 0 THEN
	    Robot.Outputs.MotionControl.SetPoint := TRUE;
	END_IF;

	(* To send _Move, send _Move ID *)
	IF NOT Buffered AND NOT Sent THEN
	    
	    Robot.Outputs.MotionCommand.MoveCommand	:= EnumToNum(Meca500Cmd#MoveLinVelTrf);
	    Robot.Outputs.MotionCommand.MoveSubIndex001 := Output_Params[1];
		Robot.Outputs.MotionCommand.MoveSubIndex002 := Output_Params[2];
		Robot.Outputs.MotionCommand.MoveSubIndex003 := Output_Params[3];
		Robot.Outputs.MotionCommand.MoveSubIndex004 := Output_Params[4];
		Robot.Outputs.MotionCommand.MoveSubIndex005 := Output_Params[5];
		Robot.Outputs.MotionCommand.MoveSubIndex006 := Output_Params[6];
	    
	    IF ExternalStateControl THEN
	        IF ExternalMoveID <> 0 AND ExternalMoveID <> 32230 AND ExternalMoveID <> 32231 THEN
	            Robot.Outputs.MotionControl.MoveID := ExternalMoveID;
	            Sent := TRUE;
	        END_IF;
	        
	    ELSE (*Not External Control*)
	        IF Robot.Outputs.MotionControl.MoveID = 32230 THEN
	            Robot.Outputs.MotionControl.MoveID := 32231;
	        ELSIF Robot.Outputs.MotionControl.MoveID = 32231 THEN
	            Robot.Outputs.MotionControl.MoveID := 32230;
	        ELSIF Robot.Outputs.MotionControl.MoveID <> 32230 OR Robot.Outputs.MotionControl.MoveID <> 32231 THEN
	            Robot.Outputs.MotionControl.MoveID := 32230;
	        END_IF;
	        Sent := TRUE;
	    END_IF;
	END_IF;

	(* Check if command has been sent, if so, check if it was received *)
	IF Sent AND
	    Robot.Outputs.MotionCommand.MoveCommand = EnumToNum(Meca500Cmd#MoveLinVelTrf) AND
	    Robot.Outputs.MotionCommand.MoveSubIndex001 = Output_Params[1] AND 
		Robot.Outputs.MotionCommand.MoveSubIndex002 = Output_Params[2] AND 
		Robot.Outputs.MotionCommand.MoveSubIndex003 = Output_Params[3] AND 
		Robot.Outputs.MotionCommand.MoveSubIndex004 = Output_Params[4] AND 
		Robot.Outputs.MotionCommand.MoveSubIndex005 = Output_Params[5] AND 
		Robot.Outputs.MotionCommand.MoveSubIndex006 = Output_Params[6] AND
		Robot.Inputs.Motion.MoveID = Robot.Outputs.MotionControl.MoveID 
	THEN
		 Buffered := TRUE;
	END_IF;


	(*If External _Move ID is equal to Internal, raise an error*)
	IF ExternalMoveID = 32230 OR ExternalMoveID = 32231 THEN
	    Error := TRUE;
	END_IF;

	FirstScan := TRUE;
ELSE
	FirstScan := False;
	Sent := FALSE;
	Buffered := FALSE;
END_IF;
END_FUNCTION_BLOCK

FUNCTION_BLOCK Meca500_MoveLinVelWRF
VAR
    Output_Params : array[1..6] of real;
    FirstScan : BOOL := False;
END_VAR
VAR_INPUT
    Execute : BOOL;
    X_Vel : REAL;
    Y_Vel : REAL;
    Z_Vel : REAL;
    rX_AngleVel : REAL;
    rY_AngleVel : REAL;
    rZ_AngleVel : REAL;
END_VAR
VAR_OUTPUT
    Sent : BOOL;
    Buffered : BOOL;
    Error : BOOL;
END_VAR
VAR_IN_OUT
    Robot : Meca500;
END_VAR
VAR_INPUT
    ExternalStateControl : BOOL;
    ExternalMoveID : UINT;
END_VAR
IF Execute THEN	
	(*Collect Inputs and store them locally*)
	Output_Params[1]:=X_Vel;
	Output_Params[2]:=Y_Vel;
	Output_Params[3]:=Z_Vel;
	Output_Params[4]:=rX_AngleVel;
	Output_Params[5]:=rY_AngleVel;
	Output_Params[6]:=rZ_AngleVel;

	(* If Values have change, Reinitialise Outputs*)

	IF FirstScan=0 OR 
		Robot.Outputs.MotionCommand.MoveSubIndex001 <> Output_Params[1] OR 
		Robot.Outputs.MotionCommand.MoveSubIndex002 <> Output_Params[2] OR 
		Robot.Outputs.MotionCommand.MoveSubIndex003 <> Output_Params[3] OR
		Robot.Outputs.MotionCommand.MoveSubIndex004 <> Output_Params[4] OR 
		Robot.Outputs.MotionCommand.MoveSubIndex005 <> Output_Params[5] OR 
		Robot.Outputs.MotionCommand.MoveSubIndex006 <> Output_Params[6] 
	THEN
		Buffered := FALSE;
		Sent := FALSE;
	END_IF;


	(*if not in legacy mode, Act Setpoint*)
	IF Robot.Outputs.MotionControl.MoveID <> 0 THEN
	    Robot.Outputs.MotionControl.SetPoint := TRUE;
	END_IF;

	(* To send _Move, send _Move ID *)
	IF NOT Buffered AND NOT Sent THEN
	    
	    Robot.Outputs.MotionCommand.MoveCommand	:= EnumToNum(Meca500Cmd#MoveLinVelWrf);
	    Robot.Outputs.MotionCommand.MoveSubIndex001 := Output_Params[1];
		Robot.Outputs.MotionCommand.MoveSubIndex002 := Output_Params[2];
		Robot.Outputs.MotionCommand.MoveSubIndex003 := Output_Params[3];
		Robot.Outputs.MotionCommand.MoveSubIndex004 := Output_Params[4];
		Robot.Outputs.MotionCommand.MoveSubIndex005 := Output_Params[5];
		Robot.Outputs.MotionCommand.MoveSubIndex006 := Output_Params[6];
	    
	    IF ExternalStateControl THEN
	        IF ExternalMoveID <> 0 AND ExternalMoveID <> 32220 AND ExternalMoveID <> 32221 THEN
	            Robot.Outputs.MotionControl.MoveID := ExternalMoveID;
	            Sent := TRUE;
	        END_IF;
	        
	    ELSE (*Not External Control*)
	        IF Robot.Outputs.MotionControl.MoveID = 32220 THEN
	            Robot.Outputs.MotionControl.MoveID := 32221;
	        ELSIF Robot.Outputs.MotionControl.MoveID = 32221 THEN
	            Robot.Outputs.MotionControl.MoveID := 32220;
	        ELSIF Robot.Outputs.MotionControl.MoveID <> 32220 OR Robot.Outputs.MotionControl.MoveID <> 32221 THEN
	            Robot.Outputs.MotionControl.MoveID := 32220;
	        END_IF;
	        Sent := TRUE;
	    END_IF;
	END_IF;

	(* Check if command has been sent, if so, check if it was received *)
	IF Sent AND
	    Robot.Outputs.MotionCommand.MoveCommand = EnumToNum(Meca500Cmd#MoveLinVelWrf) AND
	    Robot.Outputs.MotionCommand.MoveSubIndex001 = Output_Params[1] AND 
		Robot.Outputs.MotionCommand.MoveSubIndex002 = Output_Params[2] AND 
		Robot.Outputs.MotionCommand.MoveSubIndex003 = Output_Params[3] AND 
		Robot.Outputs.MotionCommand.MoveSubIndex004 = Output_Params[4] AND 
		Robot.Outputs.MotionCommand.MoveSubIndex005 = Output_Params[5] AND 
		Robot.Outputs.MotionCommand.MoveSubIndex006 = Output_Params[6] AND
		Robot.Inputs.Motion.MoveID = Robot.Outputs.MotionControl.MoveID 
	THEN
		 Buffered := TRUE;
	END_IF;


	(*If External _Move ID is equal to Internal, raise an error*)
	IF ExternalMoveID = 32220 OR ExternalMoveID = 32221 THEN
	    Error := TRUE;
	END_IF;

	FirstScan := TRUE;
ELSE
	FirstScan := False;
	Sent := FALSE;
	Buffered := FALSE;
END_IF;
END_FUNCTION_BLOCK

FUNCTION_BLOCK Meca500_MovePose
VAR
    Output_Params : array[1..6] of real;
    FirstScan : BOOL := False;
END_VAR
VAR_INPUT
    Execute : BOOL;
    Pose_X_Pos : REAL;
    Pose_Y_Pos : REAL;
    Pose_Z_Pos : REAL;
    Pose_rX_Angle : REAL;
    Pose_rY_Angle : REAL;
    Pose_rZ_Angle : REAL;
END_VAR
VAR_OUTPUT
    Sent : BOOL;
    Buffered : BOOL;
    Error : BOOL;
END_VAR
VAR_IN_OUT
    Robot : Meca500;
END_VAR
VAR_INPUT
    ExternalStateControl : BOOL;
    ExternalMoveID : UINT;
END_VAR
IF Execute THEN	
	(*Collect Inputs and store them locally*)
	Output_Params[1]:=Pose_X_Pos;
	Output_Params[2]:=Pose_Y_Pos;
	Output_Params[3]:=Pose_Z_Pos;
	Output_Params[4]:=Pose_rX_Angle;
	Output_Params[5]:=Pose_rY_Angle;
	Output_Params[6]:=Pose_rZ_Angle;

	(* If Values have change, Reinitialise Outputs*)

	IF FirstScan=0 OR 
		Robot.Outputs.MotionCommand.MoveSubIndex001 <> Output_Params[1] OR 
		Robot.Outputs.MotionCommand.MoveSubIndex002 <> Output_Params[2] OR 
		Robot.Outputs.MotionCommand.MoveSubIndex003 <> Output_Params[3] OR
		Robot.Outputs.MotionCommand.MoveSubIndex004 <> Output_Params[4] OR 
		Robot.Outputs.MotionCommand.MoveSubIndex005 <> Output_Params[5] OR 
		Robot.Outputs.MotionCommand.MoveSubIndex006 <> Output_Params[6] 
	THEN
		Buffered := FALSE;
		Sent := FALSE;
	END_IF;


	(*if not in legacy mode, Act Setpoint*)
	IF Robot.Outputs.MotionControl.MoveID <> 0 THEN
	    Robot.Outputs.MotionControl.SetPoint := TRUE;
	END_IF;

	(* To send _Move, send _Move ID *)
	IF NOT Buffered AND NOT Sent THEN
	    
	    Robot.Outputs.MotionCommand.MoveCommand	:= EnumToNum(Meca500Cmd#MovePose);
	    Robot.Outputs.MotionCommand.MoveSubIndex001 := Output_Params[1];
		Robot.Outputs.MotionCommand.MoveSubIndex002 := Output_Params[2];
		Robot.Outputs.MotionCommand.MoveSubIndex003 := Output_Params[3];
		Robot.Outputs.MotionCommand.MoveSubIndex004 := Output_Params[4];
		Robot.Outputs.MotionCommand.MoveSubIndex005 := Output_Params[5];
		Robot.Outputs.MotionCommand.MoveSubIndex006 := Output_Params[6];
	    
	    IF ExternalStateControl THEN
	        IF ExternalMoveID <> 0 AND ExternalMoveID <> 32020 AND ExternalMoveID <> 32021 THEN
	            Robot.Outputs.MotionControl.MoveID := ExternalMoveID;
	            Sent := TRUE;
	        END_IF;
	        
	    ELSE (*Not External Control*)
	        IF Robot.Outputs.MotionControl.MoveID = 32020 THEN
	            Robot.Outputs.MotionControl.MoveID := 32021;
	        ELSIF Robot.Outputs.MotionControl.MoveID = 32021 THEN
	            Robot.Outputs.MotionControl.MoveID := 32020;
	        ELSIF Robot.Outputs.MotionControl.MoveID <> 32020 OR Robot.Outputs.MotionControl.MoveID <> 32021 THEN
	            Robot.Outputs.MotionControl.MoveID := 32020;
	        END_IF;
	        Sent := TRUE;
	    END_IF;
	END_IF;

	(* Check if command has been sent, if so, check if it was received *)
	IF Sent AND
	    Robot.Outputs.MotionCommand.MoveCommand = EnumToNum(Meca500Cmd#MovePose) AND
	    Robot.Outputs.MotionCommand.MoveSubIndex001 = Output_Params[1] AND 
		Robot.Outputs.MotionCommand.MoveSubIndex002 = Output_Params[2] AND 
		Robot.Outputs.MotionCommand.MoveSubIndex003 = Output_Params[3] AND 
		Robot.Outputs.MotionCommand.MoveSubIndex004 = Output_Params[4] AND 
		Robot.Outputs.MotionCommand.MoveSubIndex005 = Output_Params[5] AND 
		Robot.Outputs.MotionCommand.MoveSubIndex006 = Output_Params[6] AND
		Robot.Inputs.Motion.MoveID = Robot.Outputs.MotionControl.MoveID 
	THEN
		 Buffered := TRUE;
	END_IF;


	(*If External _Move ID is equal to Internal, raise an error*)
	IF ExternalMoveID = 32020 OR ExternalMoveID = 32021 THEN
	    Error := TRUE;
	END_IF;

	FirstScan := TRUE;
ELSE
	FirstScan := False;
	Sent := FALSE;
	Buffered := FALSE;
END_IF;
END_FUNCTION_BLOCK

FUNCTION_BLOCK Meca500_SetAutoConf
VAR
    Output_Params : array[1..6] of real;
    FirstScan : BOOL := False;
END_VAR
VAR_INPUT
    Execute : BOOL;
    Enable : REAL;
END_VAR
VAR_OUTPUT
    Sent : BOOL;
    Buffered : BOOL;
    Error : BOOL;
END_VAR
VAR_IN_OUT
    Robot : Meca500;
END_VAR
VAR_INPUT
    ExternalStateControl : BOOL;
    ExternalMoveID : UINT;
END_VAR
IF Execute THEN	
	(*Collect Inputs and store them locally*)
	Output_Params[1]:=Enable;
	Output_Params[2]:=0;
	Output_Params[3]:=0;
	Output_Params[4]:=0;
	Output_Params[5]:=0;
	Output_Params[6]:=0;

	(* If Values have change, Reinitialise Outputs*)

	IF FirstScan=0 OR 
		Robot.Outputs.MotionCommand.MoveSubIndex001 <> Output_Params[1] OR 
		Robot.Outputs.MotionCommand.MoveSubIndex002 <> Output_Params[2] OR 
		Robot.Outputs.MotionCommand.MoveSubIndex003 <> Output_Params[3] OR
		Robot.Outputs.MotionCommand.MoveSubIndex004 <> Output_Params[4] OR 
		Robot.Outputs.MotionCommand.MoveSubIndex005 <> Output_Params[5] OR 
		Robot.Outputs.MotionCommand.MoveSubIndex006 <> Output_Params[6] 
	THEN
		Buffered := FALSE;
		Sent := FALSE;
	END_IF;


	(*if not in legacy mode, Act Setpoint*)
	IF Robot.Outputs.MotionControl.MoveID <> 0 THEN
	    Robot.Outputs.MotionControl.SetPoint := TRUE;
	END_IF;

	(* To send _Move, send _Move ID *)
	IF NOT Buffered AND NOT Sent THEN
	    
	    Robot.Outputs.MotionCommand.MoveCommand	:= EnumToNum(Meca500Cmd#SetAutoConf);
	    Robot.Outputs.MotionCommand.MoveSubIndex001 := Output_Params[1];
		Robot.Outputs.MotionCommand.MoveSubIndex002 := Output_Params[2];
		Robot.Outputs.MotionCommand.MoveSubIndex003 := Output_Params[3];
		Robot.Outputs.MotionCommand.MoveSubIndex004 := Output_Params[4];
		Robot.Outputs.MotionCommand.MoveSubIndex005 := Output_Params[5];
		Robot.Outputs.MotionCommand.MoveSubIndex006 := Output_Params[6];
	    
	    IF ExternalStateControl THEN
	        IF ExternalMoveID <> 0 AND ExternalMoveID <> 32160 AND ExternalMoveID <> 32161 THEN
	            Robot.Outputs.MotionControl.MoveID := ExternalMoveID;
	            Sent := TRUE;
	        END_IF;
	        
	    ELSE (*Not External Control*)
	        IF Robot.Outputs.MotionControl.MoveID = 32160 THEN
	            Robot.Outputs.MotionControl.MoveID := 32161;
	        ELSIF Robot.Outputs.MotionControl.MoveID = 32161 THEN
	            Robot.Outputs.MotionControl.MoveID := 32160;
	        ELSIF Robot.Outputs.MotionControl.MoveID <> 32160 OR Robot.Outputs.MotionControl.MoveID <> 32161 THEN
	            Robot.Outputs.MotionControl.MoveID := 32160;
	        END_IF;
	        Sent := TRUE;
	    END_IF;
	END_IF;

	(* Check if command has been sent, if so, check if it was received *)
	IF Sent AND
	    Robot.Outputs.MotionCommand.MoveCommand = EnumToNum(Meca500Cmd#SetAutoConf) AND
	    Robot.Outputs.MotionCommand.MoveSubIndex001 = Output_Params[1] AND 
		Robot.Outputs.MotionCommand.MoveSubIndex002 = Output_Params[2] AND 
		Robot.Outputs.MotionCommand.MoveSubIndex003 = Output_Params[3] AND 
		Robot.Outputs.MotionCommand.MoveSubIndex004 = Output_Params[4] AND 
		Robot.Outputs.MotionCommand.MoveSubIndex005 = Output_Params[5] AND 
		Robot.Outputs.MotionCommand.MoveSubIndex006 = Output_Params[6] AND
		Robot.Inputs.Motion.MoveID = Robot.Outputs.MotionControl.MoveID 
	THEN
		 Buffered := TRUE;
	END_IF;


	(*If External _Move ID is equal to Internal, raise an error*)
	IF ExternalMoveID = 32160 OR ExternalMoveID = 32161 THEN
	    Error := TRUE;
	END_IF;

	FirstScan := TRUE;
ELSE
	FirstScan := False;
	Sent := FALSE;
	Buffered := FALSE;
END_IF;
END_FUNCTION_BLOCK

FUNCTION_BLOCK Meca500_SetAutoConfTurn
VAR
    Output_Params : array[1..6] of real;
    FirstScan : BOOL := False;
END_VAR
VAR_INPUT
    Execute : BOOL;
    Enable : REAL;
END_VAR
VAR_OUTPUT
    Sent : BOOL;
    Buffered : BOOL;
    Error : BOOL;
END_VAR
VAR_IN_OUT
    Robot : Meca500;
END_VAR
VAR_INPUT
    ExternalStateControl : BOOL;
    ExternalMoveID : UINT;
END_VAR
IF Execute THEN	
	(*Collect Inputs and store them locally*)
	Output_Params[1]:=Enable;
	Output_Params[2]:=0;
	Output_Params[3]:=0;
	Output_Params[4]:=0;
	Output_Params[5]:=0;
	Output_Params[6]:=0;

	(* If Values have change, Reinitialise Outputs*)

	IF FirstScan=0 OR 
		Robot.Outputs.MotionCommand.MoveSubIndex001 <> Output_Params[1] OR 
		Robot.Outputs.MotionCommand.MoveSubIndex002 <> Output_Params[2] OR 
		Robot.Outputs.MotionCommand.MoveSubIndex003 <> Output_Params[3] OR
		Robot.Outputs.MotionCommand.MoveSubIndex004 <> Output_Params[4] OR 
		Robot.Outputs.MotionCommand.MoveSubIndex005 <> Output_Params[5] OR 
		Robot.Outputs.MotionCommand.MoveSubIndex006 <> Output_Params[6] 
	THEN
		Buffered := FALSE;
		Sent := FALSE;
	END_IF;


	(*if not in legacy mode, Act Setpoint*)
	IF Robot.Outputs.MotionControl.MoveID <> 0 THEN
	    Robot.Outputs.MotionControl.SetPoint := TRUE;
	END_IF;

	(* To send _Move, send _Move ID *)
	IF NOT Buffered AND NOT Sent THEN
	    
	    Robot.Outputs.MotionCommand.MoveCommand	:= EnumToNum(Meca500Cmd#SetAutoConfTurn);
	    Robot.Outputs.MotionCommand.MoveSubIndex001 := Output_Params[1];
		Robot.Outputs.MotionCommand.MoveSubIndex002 := Output_Params[2];
		Robot.Outputs.MotionCommand.MoveSubIndex003 := Output_Params[3];
		Robot.Outputs.MotionCommand.MoveSubIndex004 := Output_Params[4];
		Robot.Outputs.MotionCommand.MoveSubIndex005 := Output_Params[5];
		Robot.Outputs.MotionCommand.MoveSubIndex006 := Output_Params[6];
	    
	    IF ExternalStateControl THEN
	        IF ExternalMoveID <> 0 AND ExternalMoveID <> 32260 AND ExternalMoveID <> 32261 THEN
	            Robot.Outputs.MotionControl.MoveID := ExternalMoveID;
	            Sent := TRUE;
	        END_IF;
	        
	    ELSE (*Not External Control*)
	        IF Robot.Outputs.MotionControl.MoveID = 32260 THEN
	            Robot.Outputs.MotionControl.MoveID := 32261;
	        ELSIF Robot.Outputs.MotionControl.MoveID = 32261 THEN
	            Robot.Outputs.MotionControl.MoveID := 32260;
	        ELSIF Robot.Outputs.MotionControl.MoveID <> 32260 OR Robot.Outputs.MotionControl.MoveID <> 32261 THEN
	            Robot.Outputs.MotionControl.MoveID := 32260;
	        END_IF;
	        Sent := TRUE;
	    END_IF;
	END_IF;

	(* Check if command has been sent, if so, check if it was received *)
	IF Sent AND
	    Robot.Outputs.MotionCommand.MoveCommand = EnumToNum(Meca500Cmd#SetAutoConfTurn) AND
	    Robot.Outputs.MotionCommand.MoveSubIndex001 = Output_Params[1] AND 
		Robot.Outputs.MotionCommand.MoveSubIndex002 = Output_Params[2] AND 
		Robot.Outputs.MotionCommand.MoveSubIndex003 = Output_Params[3] AND 
		Robot.Outputs.MotionCommand.MoveSubIndex004 = Output_Params[4] AND 
		Robot.Outputs.MotionCommand.MoveSubIndex005 = Output_Params[5] AND 
		Robot.Outputs.MotionCommand.MoveSubIndex006 = Output_Params[6] AND
		Robot.Inputs.Motion.MoveID = Robot.Outputs.MotionControl.MoveID 
	THEN
		 Buffered := TRUE;
	END_IF;


	(*If External _Move ID is equal to Internal, raise an error*)
	IF ExternalMoveID = 32260 OR ExternalMoveID = 32261 THEN
	    Error := TRUE;
	END_IF;

	FirstScan := TRUE;
ELSE
	FirstScan := False;
	Sent := FALSE;
	Buffered := FALSE;
END_IF;
END_FUNCTION_BLOCK

FUNCTION_BLOCK Meca500_SetBlending
VAR
    Output_Params : array[1..6] of real;
    FirstScan : BOOL := False;
END_VAR
VAR_INPUT
    Execute : BOOL;
    Blending_Percentage : REAL;
END_VAR
VAR_OUTPUT
    Sent : BOOL;
    Buffered : BOOL;
    Error : BOOL;
END_VAR
VAR_IN_OUT
    Robot : Meca500;
END_VAR
VAR_INPUT
    ExternalStateControl : BOOL;
    ExternalMoveID : UINT;
END_VAR
IF Execute THEN	
	(*Collect Inputs and store them locally*)
	Output_Params[1]:=Blending_Percentage;
	Output_Params[2]:=0;
	Output_Params[3]:=0;
	Output_Params[4]:=0;
	Output_Params[5]:=0;
	Output_Params[6]:=0;

	(* If Values have change, Reinitialise Outputs*)

	IF FirstScan=0 OR 
		Robot.Outputs.MotionCommand.MoveSubIndex001 <> Output_Params[1] OR 
		Robot.Outputs.MotionCommand.MoveSubIndex002 <> Output_Params[2] OR 
		Robot.Outputs.MotionCommand.MoveSubIndex003 <> Output_Params[3] OR
		Robot.Outputs.MotionCommand.MoveSubIndex004 <> Output_Params[4] OR 
		Robot.Outputs.MotionCommand.MoveSubIndex005 <> Output_Params[5] OR 
		Robot.Outputs.MotionCommand.MoveSubIndex006 <> Output_Params[6] 
	THEN
		Buffered := FALSE;
		Sent := FALSE;
	END_IF;


	(*if not in legacy mode, Act Setpoint*)
	IF Robot.Outputs.MotionControl.MoveID <> 0 THEN
	    Robot.Outputs.MotionControl.SetPoint := TRUE;
	END_IF;

	(* To send _Move, send _Move ID *)
	IF NOT Buffered AND NOT Sent THEN
	    
	    Robot.Outputs.MotionCommand.MoveCommand	:= EnumToNum(Meca500Cmd#SetBlending);
	    Robot.Outputs.MotionCommand.MoveSubIndex001 := Output_Params[1];
		Robot.Outputs.MotionCommand.MoveSubIndex002 := Output_Params[2];
		Robot.Outputs.MotionCommand.MoveSubIndex003 := Output_Params[3];
		Robot.Outputs.MotionCommand.MoveSubIndex004 := Output_Params[4];
		Robot.Outputs.MotionCommand.MoveSubIndex005 := Output_Params[5];
		Robot.Outputs.MotionCommand.MoveSubIndex006 := Output_Params[6];
	    
	    IF ExternalStateControl THEN
	        IF ExternalMoveID <> 0 AND ExternalMoveID <> 32070 AND ExternalMoveID <> 32071 THEN
	            Robot.Outputs.MotionControl.MoveID := ExternalMoveID;
	            Sent := TRUE;
	        END_IF;
	        
	    ELSE (*Not External Control*)
	        IF Robot.Outputs.MotionControl.MoveID = 32070 THEN
	            Robot.Outputs.MotionControl.MoveID := 32071;
	        ELSIF Robot.Outputs.MotionControl.MoveID = 32071 THEN
	            Robot.Outputs.MotionControl.MoveID := 32070;
	        ELSIF Robot.Outputs.MotionControl.MoveID <> 32070 OR Robot.Outputs.MotionControl.MoveID <> 32071 THEN
	            Robot.Outputs.MotionControl.MoveID := 32070;
	        END_IF;
	        Sent := TRUE;
	    END_IF;
	END_IF;

	(* Check if command has been sent, if so, check if it was received *)
	IF Sent AND
	    Robot.Outputs.MotionCommand.MoveCommand = EnumToNum(Meca500Cmd#SetBlending) AND
	    Robot.Outputs.MotionCommand.MoveSubIndex001 = Output_Params[1] AND 
		Robot.Outputs.MotionCommand.MoveSubIndex002 = Output_Params[2] AND 
		Robot.Outputs.MotionCommand.MoveSubIndex003 = Output_Params[3] AND 
		Robot.Outputs.MotionCommand.MoveSubIndex004 = Output_Params[4] AND 
		Robot.Outputs.MotionCommand.MoveSubIndex005 = Output_Params[5] AND 
		Robot.Outputs.MotionCommand.MoveSubIndex006 = Output_Params[6] AND
		Robot.Inputs.Motion.MoveID = Robot.Outputs.MotionControl.MoveID 
	THEN
		 Buffered := TRUE;
	END_IF;


	(*If External _Move ID is equal to Internal, raise an error*)
	IF ExternalMoveID = 32070 OR ExternalMoveID = 32071 THEN
	    Error := TRUE;
	END_IF;

	FirstScan := TRUE;
ELSE
	FirstScan := False;
	Sent := FALSE;
	Buffered := FALSE;
END_IF;
END_FUNCTION_BLOCK

FUNCTION_BLOCK Meca500_SetCartAcc
VAR
    Output_Params : array[1..6] of real;
    FirstScan : BOOL := False;
END_VAR
VAR_INPUT
    Execute : BOOL;
    Acceleration_Percentage : REAL;
END_VAR
VAR_OUTPUT
    Sent : BOOL;
    Buffered : BOOL;
    Error : BOOL;
END_VAR
VAR_IN_OUT
    Robot : Meca500;
END_VAR
VAR_INPUT
    ExternalStateControl : BOOL;
    ExternalMoveID : UINT;
END_VAR
IF Execute THEN	
	(*Collect Inputs and store them locally*)
	Output_Params[1]:=Acceleration_Percentage;
	Output_Params[2]:=0;
	Output_Params[3]:=0;
	Output_Params[4]:=0;
	Output_Params[5]:=0;
	Output_Params[6]:=0;

	(* If Values have change, Reinitialise Outputs*)

	IF FirstScan=0 OR 
		Robot.Outputs.MotionCommand.MoveSubIndex001 <> Output_Params[1] OR 
		Robot.Outputs.MotionCommand.MoveSubIndex002 <> Output_Params[2] OR 
		Robot.Outputs.MotionCommand.MoveSubIndex003 <> Output_Params[3] OR
		Robot.Outputs.MotionCommand.MoveSubIndex004 <> Output_Params[4] OR 
		Robot.Outputs.MotionCommand.MoveSubIndex005 <> Output_Params[5] OR 
		Robot.Outputs.MotionCommand.MoveSubIndex006 <> Output_Params[6] 
	THEN
		Buffered := FALSE;
		Sent := FALSE;
	END_IF;


	(*if not in legacy mode, Act Setpoint*)
	IF Robot.Outputs.MotionControl.MoveID <> 0 THEN
	    Robot.Outputs.MotionControl.SetPoint := TRUE;
	END_IF;

	(* To send _Move, send _Move ID *)
	IF NOT Buffered AND NOT Sent THEN
	    
	    Robot.Outputs.MotionCommand.MoveCommand	:= EnumToNum(Meca500Cmd#SetCartAcc);
	    Robot.Outputs.MotionCommand.MoveSubIndex001 := Output_Params[1];
		Robot.Outputs.MotionCommand.MoveSubIndex002 := Output_Params[2];
		Robot.Outputs.MotionCommand.MoveSubIndex003 := Output_Params[3];
		Robot.Outputs.MotionCommand.MoveSubIndex004 := Output_Params[4];
		Robot.Outputs.MotionCommand.MoveSubIndex005 := Output_Params[5];
		Robot.Outputs.MotionCommand.MoveSubIndex006 := Output_Params[6];
	    
	    IF ExternalStateControl THEN
	        IF ExternalMoveID <> 0 AND ExternalMoveID <> 32120 AND ExternalMoveID <> 32121 THEN
	            Robot.Outputs.MotionControl.MoveID := ExternalMoveID;
	            Sent := TRUE;
	        END_IF;
	        
	    ELSE (*Not External Control*)
	        IF Robot.Outputs.MotionControl.MoveID = 32120 THEN
	            Robot.Outputs.MotionControl.MoveID := 32121;
	        ELSIF Robot.Outputs.MotionControl.MoveID = 32121 THEN
	            Robot.Outputs.MotionControl.MoveID := 32120;
	        ELSIF Robot.Outputs.MotionControl.MoveID <> 32120 OR Robot.Outputs.MotionControl.MoveID <> 32121 THEN
	            Robot.Outputs.MotionControl.MoveID := 32120;
	        END_IF;
	        Sent := TRUE;
	    END_IF;
	END_IF;

	(* Check if command has been sent, if so, check if it was received *)
	IF Sent AND
	    Robot.Outputs.MotionCommand.MoveCommand = EnumToNum(Meca500Cmd#SetCartAcc) AND
	    Robot.Outputs.MotionCommand.MoveSubIndex001 = Output_Params[1] AND 
		Robot.Outputs.MotionCommand.MoveSubIndex002 = Output_Params[2] AND 
		Robot.Outputs.MotionCommand.MoveSubIndex003 = Output_Params[3] AND 
		Robot.Outputs.MotionCommand.MoveSubIndex004 = Output_Params[4] AND 
		Robot.Outputs.MotionCommand.MoveSubIndex005 = Output_Params[5] AND 
		Robot.Outputs.MotionCommand.MoveSubIndex006 = Output_Params[6] AND
		Robot.Inputs.Motion.MoveID = Robot.Outputs.MotionControl.MoveID 
	THEN
		 Buffered := TRUE;
	END_IF;


	(*If External _Move ID is equal to Internal, raise an error*)
	IF ExternalMoveID = 32120 OR ExternalMoveID = 32121 THEN
	    Error := TRUE;
	END_IF;

	FirstScan := TRUE;
ELSE
	FirstScan := False;
	Sent := FALSE;
	Buffered := FALSE;
END_IF;
END_FUNCTION_BLOCK

FUNCTION_BLOCK Meca500_SetCartAngVel
VAR
    Output_Params : array[1..6] of real;
    FirstScan : BOOL := False;
END_VAR
VAR_INPUT
    Execute : BOOL;
    Velocity_Limit : REAL;
END_VAR
VAR_OUTPUT
    Sent : BOOL;
    Buffered : BOOL;
    Error : BOOL;
END_VAR
VAR_IN_OUT
    Robot : Meca500;
END_VAR
VAR_INPUT
    ExternalStateControl : BOOL;
    ExternalMoveID : UINT;
END_VAR
IF Execute THEN	
	(*Collect Inputs and store them locally*)
	Output_Params[1]:=Velocity_Limit;
	Output_Params[2]:=0;
	Output_Params[3]:=0;
	Output_Params[4]:=0;
	Output_Params[5]:=0;
	Output_Params[6]:=0;

	(* If Values have change, Reinitialise Outputs*)

	IF FirstScan=0 OR 
		Robot.Outputs.MotionCommand.MoveSubIndex001 <> Output_Params[1] OR 
		Robot.Outputs.MotionCommand.MoveSubIndex002 <> Output_Params[2] OR 
		Robot.Outputs.MotionCommand.MoveSubIndex003 <> Output_Params[3] OR
		Robot.Outputs.MotionCommand.MoveSubIndex004 <> Output_Params[4] OR 
		Robot.Outputs.MotionCommand.MoveSubIndex005 <> Output_Params[5] OR 
		Robot.Outputs.MotionCommand.MoveSubIndex006 <> Output_Params[6] 
	THEN
		Buffered := FALSE;
		Sent := FALSE;
	END_IF;


	(*if not in legacy mode, Act Setpoint*)
	IF Robot.Outputs.MotionControl.MoveID <> 0 THEN
	    Robot.Outputs.MotionControl.SetPoint := TRUE;
	END_IF;

	(* To send _Move, send _Move ID *)
	IF NOT Buffered AND NOT Sent THEN
	    
	    Robot.Outputs.MotionCommand.MoveCommand	:= EnumToNum(Meca500Cmd#SetCartAngVel);
	    Robot.Outputs.MotionCommand.MoveSubIndex001 := Output_Params[1];
		Robot.Outputs.MotionCommand.MoveSubIndex002 := Output_Params[2];
		Robot.Outputs.MotionCommand.MoveSubIndex003 := Output_Params[3];
		Robot.Outputs.MotionCommand.MoveSubIndex004 := Output_Params[4];
		Robot.Outputs.MotionCommand.MoveSubIndex005 := Output_Params[5];
		Robot.Outputs.MotionCommand.MoveSubIndex006 := Output_Params[6];
	    
	    IF ExternalStateControl THEN
	        IF ExternalMoveID <> 0 AND ExternalMoveID <> 32100 AND ExternalMoveID <> 32101 THEN
	            Robot.Outputs.MotionControl.MoveID := ExternalMoveID;
	            Sent := TRUE;
	        END_IF;
	        
	    ELSE (*Not External Control*)
	        IF Robot.Outputs.MotionControl.MoveID = 32100 THEN
	            Robot.Outputs.MotionControl.MoveID := 32101;
	        ELSIF Robot.Outputs.MotionControl.MoveID = 32101 THEN
	            Robot.Outputs.MotionControl.MoveID := 32100;
	        ELSIF Robot.Outputs.MotionControl.MoveID <> 32100 OR Robot.Outputs.MotionControl.MoveID <> 32101 THEN
	            Robot.Outputs.MotionControl.MoveID := 32100;
	        END_IF;
	        Sent := TRUE;
	    END_IF;
	END_IF;

	(* Check if command has been sent, if so, check if it was received *)
	IF Sent AND
	    Robot.Outputs.MotionCommand.MoveCommand = EnumToNum(Meca500Cmd#SetCartAngVel) AND
	    Robot.Outputs.MotionCommand.MoveSubIndex001 = Output_Params[1] AND 
		Robot.Outputs.MotionCommand.MoveSubIndex002 = Output_Params[2] AND 
		Robot.Outputs.MotionCommand.MoveSubIndex003 = Output_Params[3] AND 
		Robot.Outputs.MotionCommand.MoveSubIndex004 = Output_Params[4] AND 
		Robot.Outputs.MotionCommand.MoveSubIndex005 = Output_Params[5] AND 
		Robot.Outputs.MotionCommand.MoveSubIndex006 = Output_Params[6] AND
		Robot.Inputs.Motion.MoveID = Robot.Outputs.MotionControl.MoveID 
	THEN
		 Buffered := TRUE;
	END_IF;


	(*If External _Move ID is equal to Internal, raise an error*)
	IF ExternalMoveID = 32100 OR ExternalMoveID = 32101 THEN
	    Error := TRUE;
	END_IF;

	FirstScan := TRUE;
ELSE
	FirstScan := False;
	Sent := FALSE;
	Buffered := FALSE;
END_IF;
END_FUNCTION_BLOCK

FUNCTION_BLOCK Meca500_SetCartLinVel
VAR
    Output_Params : array[1..6] of real;
    FirstScan : BOOL := False;
END_VAR
VAR_INPUT
    Execute : BOOL;
    Velocity_Limit : REAL;
END_VAR
VAR_OUTPUT
    Sent : BOOL;
    Buffered : BOOL;
    Error : BOOL;
END_VAR
VAR_IN_OUT
    Robot : Meca500;
END_VAR
VAR_INPUT
    ExternalStateControl : BOOL;
    ExternalMoveID : UINT;
END_VAR
IF Execute THEN	
	(*Collect Inputs and store them locally*)
	Output_Params[1]:=Velocity_Limit;
	Output_Params[2]:=0;
	Output_Params[3]:=0;
	Output_Params[4]:=0;
	Output_Params[5]:=0;
	Output_Params[6]:=0;

	(* If Values have change, Reinitialise Outputs*)

	IF FirstScan=0 OR 
		Robot.Outputs.MotionCommand.MoveSubIndex001 <> Output_Params[1] OR 
		Robot.Outputs.MotionCommand.MoveSubIndex002 <> Output_Params[2] OR 
		Robot.Outputs.MotionCommand.MoveSubIndex003 <> Output_Params[3] OR
		Robot.Outputs.MotionCommand.MoveSubIndex004 <> Output_Params[4] OR 
		Robot.Outputs.MotionCommand.MoveSubIndex005 <> Output_Params[5] OR 
		Robot.Outputs.MotionCommand.MoveSubIndex006 <> Output_Params[6] 
	THEN
		Buffered := FALSE;
		Sent := FALSE;
	END_IF;


	(*if not in legacy mode, Act Setpoint*)
	IF Robot.Outputs.MotionControl.MoveID <> 0 THEN
	    Robot.Outputs.MotionControl.SetPoint := TRUE;
	END_IF;

	(* To send _Move, send _Move ID *)
	IF NOT Buffered AND NOT Sent THEN
	    
	    Robot.Outputs.MotionCommand.MoveCommand	:= EnumToNum(Meca500Cmd#SetCartLinVel);
	    Robot.Outputs.MotionCommand.MoveSubIndex001 := Output_Params[1];
		Robot.Outputs.MotionCommand.MoveSubIndex002 := Output_Params[2];
		Robot.Outputs.MotionCommand.MoveSubIndex003 := Output_Params[3];
		Robot.Outputs.MotionCommand.MoveSubIndex004 := Output_Params[4];
		Robot.Outputs.MotionCommand.MoveSubIndex005 := Output_Params[5];
		Robot.Outputs.MotionCommand.MoveSubIndex006 := Output_Params[6];
	    
	    IF ExternalStateControl THEN
	        IF ExternalMoveID <> 0 AND ExternalMoveID <> 32110 AND ExternalMoveID <> 32111 THEN
	            Robot.Outputs.MotionControl.MoveID := ExternalMoveID;
	            Sent := TRUE;
	        END_IF;
	        
	    ELSE (*Not External Control*)
	        IF Robot.Outputs.MotionControl.MoveID = 32110 THEN
	            Robot.Outputs.MotionControl.MoveID := 32111;
	        ELSIF Robot.Outputs.MotionControl.MoveID = 32111 THEN
	            Robot.Outputs.MotionControl.MoveID := 32110;
	        ELSIF Robot.Outputs.MotionControl.MoveID <> 32110 OR Robot.Outputs.MotionControl.MoveID <> 32111 THEN
	            Robot.Outputs.MotionControl.MoveID := 32110;
	        END_IF;
	        Sent := TRUE;
	    END_IF;
	END_IF;

	(* Check if command has been sent, if so, check if it was received *)
	IF Sent AND
	    Robot.Outputs.MotionCommand.MoveCommand = EnumToNum(Meca500Cmd#SetCartLinVel) AND
	    Robot.Outputs.MotionCommand.MoveSubIndex001 = Output_Params[1] AND 
		Robot.Outputs.MotionCommand.MoveSubIndex002 = Output_Params[2] AND 
		Robot.Outputs.MotionCommand.MoveSubIndex003 = Output_Params[3] AND 
		Robot.Outputs.MotionCommand.MoveSubIndex004 = Output_Params[4] AND 
		Robot.Outputs.MotionCommand.MoveSubIndex005 = Output_Params[5] AND 
		Robot.Outputs.MotionCommand.MoveSubIndex006 = Output_Params[6] AND
		Robot.Inputs.Motion.MoveID = Robot.Outputs.MotionControl.MoveID 
	THEN
		 Buffered := TRUE;
	END_IF;


	(*If External _Move ID is equal to Internal, raise an error*)
	IF ExternalMoveID = 32110 OR ExternalMoveID = 32111 THEN
	    Error := TRUE;
	END_IF;

	FirstScan := TRUE;
ELSE
	FirstScan := False;
	Sent := FALSE;
	Buffered := FALSE;
END_IF;
END_FUNCTION_BLOCK

FUNCTION_BLOCK Meca500_SetCheckpoint
VAR
    Output_Params : array[1..6] of real;
    FirstScan : BOOL := False;
END_VAR
VAR_INPUT
    Execute : BOOL;
    CheckpointID : REAL;
END_VAR
VAR_OUTPUT
    Sent : BOOL;
    Buffered : BOOL;
    Error : BOOL;
END_VAR
VAR_IN_OUT
    Robot : Meca500;
END_VAR
VAR_INPUT
    ExternalStateControl : BOOL;
    ExternalMoveID : UINT;
END_VAR
IF Execute THEN	
	(*Collect Inputs and store them locally*)
	Output_Params[1]:=CheckpointID;
	Output_Params[2]:=0;
	Output_Params[3]:=0;
	Output_Params[4]:=0;
	Output_Params[5]:=0;
	Output_Params[6]:=0;

	(* If Values have change, Reinitialise Outputs*)

	IF FirstScan=0 OR 
		Robot.Outputs.MotionCommand.MoveSubIndex001 <> Output_Params[1] OR 
		Robot.Outputs.MotionCommand.MoveSubIndex002 <> Output_Params[2] OR 
		Robot.Outputs.MotionCommand.MoveSubIndex003 <> Output_Params[3] OR
		Robot.Outputs.MotionCommand.MoveSubIndex004 <> Output_Params[4] OR 
		Robot.Outputs.MotionCommand.MoveSubIndex005 <> Output_Params[5] OR 
		Robot.Outputs.MotionCommand.MoveSubIndex006 <> Output_Params[6] 
	THEN
		Buffered := FALSE;
		Sent := FALSE;
	END_IF;


	(*if not in legacy mode, Act Setpoint*)
	IF Robot.Outputs.MotionControl.MoveID <> 0 THEN
	    Robot.Outputs.MotionControl.SetPoint := TRUE;
	END_IF;

	(* To send _Move, send _Move ID *)
	IF NOT Buffered AND NOT Sent THEN
	    
	    Robot.Outputs.MotionCommand.MoveCommand	:= EnumToNum(Meca500Cmd#SetCheckpoint);
	    Robot.Outputs.MotionCommand.MoveSubIndex001 := Output_Params[1];
		Robot.Outputs.MotionCommand.MoveSubIndex002 := Output_Params[2];
		Robot.Outputs.MotionCommand.MoveSubIndex003 := Output_Params[3];
		Robot.Outputs.MotionCommand.MoveSubIndex004 := Output_Params[4];
		Robot.Outputs.MotionCommand.MoveSubIndex005 := Output_Params[5];
		Robot.Outputs.MotionCommand.MoveSubIndex006 := Output_Params[6];
	    
	    IF ExternalStateControl THEN
	        IF ExternalMoveID <> 0 AND ExternalMoveID <> 32170 AND ExternalMoveID <> 32171 THEN
	            Robot.Outputs.MotionControl.MoveID := ExternalMoveID;
	            Sent := TRUE;
	        END_IF;
	        
	    ELSE (*Not External Control*)
	        IF Robot.Outputs.MotionControl.MoveID = 32170 THEN
	            Robot.Outputs.MotionControl.MoveID := 32171;
	        ELSIF Robot.Outputs.MotionControl.MoveID = 32171 THEN
	            Robot.Outputs.MotionControl.MoveID := 32170;
	        ELSIF Robot.Outputs.MotionControl.MoveID <> 32170 OR Robot.Outputs.MotionControl.MoveID <> 32171 THEN
	            Robot.Outputs.MotionControl.MoveID := 32170;
	        END_IF;
	        Sent := TRUE;
	    END_IF;
	END_IF;

	(* Check if command has been sent, if so, check if it was received *)
	IF Sent AND
	    Robot.Outputs.MotionCommand.MoveCommand = EnumToNum(Meca500Cmd#SetCheckpoint) AND
	    Robot.Outputs.MotionCommand.MoveSubIndex001 = Output_Params[1] AND 
		Robot.Outputs.MotionCommand.MoveSubIndex002 = Output_Params[2] AND 
		Robot.Outputs.MotionCommand.MoveSubIndex003 = Output_Params[3] AND 
		Robot.Outputs.MotionCommand.MoveSubIndex004 = Output_Params[4] AND 
		Robot.Outputs.MotionCommand.MoveSubIndex005 = Output_Params[5] AND 
		Robot.Outputs.MotionCommand.MoveSubIndex006 = Output_Params[6] AND
		Robot.Inputs.Motion.MoveID = Robot.Outputs.MotionControl.MoveID 
	THEN
		 Buffered := TRUE;
	END_IF;


	(*If External _Move ID is equal to Internal, raise an error*)
	IF ExternalMoveID = 32170 OR ExternalMoveID = 32171 THEN
	    Error := TRUE;
	END_IF;

	FirstScan := TRUE;
ELSE
	FirstScan := False;
	Sent := FALSE;
	Buffered := FALSE;
END_IF;
END_FUNCTION_BLOCK

FUNCTION_BLOCK Meca500_SetConf
VAR
    Output_Params : array[1..6] of real;
    FirstScan : BOOL := False;
END_VAR
VAR_INPUT
    Execute : BOOL;
    Shoulder : REAL;
    Elbow : REAL;
    Wrist : REAL;
END_VAR
VAR_OUTPUT
    Sent : BOOL;
    Buffered : BOOL;
    Error : BOOL;
END_VAR
VAR_IN_OUT
    Robot : Meca500;
END_VAR
VAR_INPUT
    ExternalStateControl : BOOL;
    ExternalMoveID : UINT;
END_VAR
IF Execute THEN	
	(*Collect Inputs and store them locally*)
	Output_Params[1]:=Shoulder;
	Output_Params[2]:=Elbow;
	Output_Params[3]:=Wrist;
	Output_Params[4]:=0;
	Output_Params[5]:=0;
	Output_Params[6]:=0;

	(* If Values have change, Reinitialise Outputs*)

	IF FirstScan=0 OR 
		Robot.Outputs.MotionCommand.MoveSubIndex001 <> Output_Params[1] OR 
		Robot.Outputs.MotionCommand.MoveSubIndex002 <> Output_Params[2] OR 
		Robot.Outputs.MotionCommand.MoveSubIndex003 <> Output_Params[3] OR
		Robot.Outputs.MotionCommand.MoveSubIndex004 <> Output_Params[4] OR 
		Robot.Outputs.MotionCommand.MoveSubIndex005 <> Output_Params[5] OR 
		Robot.Outputs.MotionCommand.MoveSubIndex006 <> Output_Params[6] 
	THEN
		Buffered := FALSE;
		Sent := FALSE;
	END_IF;


	(*if not in legacy mode, Act Setpoint*)
	IF Robot.Outputs.MotionControl.MoveID <> 0 THEN
	    Robot.Outputs.MotionControl.SetPoint := TRUE;
	END_IF;

	(* To send _Move, send _Move ID *)
	IF NOT Buffered AND NOT Sent THEN
	    
	    Robot.Outputs.MotionCommand.MoveCommand	:= EnumToNum(Meca500Cmd#SetConf);
	    Robot.Outputs.MotionCommand.MoveSubIndex001 := Output_Params[1];
		Robot.Outputs.MotionCommand.MoveSubIndex002 := Output_Params[2];
		Robot.Outputs.MotionCommand.MoveSubIndex003 := Output_Params[3];
		Robot.Outputs.MotionCommand.MoveSubIndex004 := Output_Params[4];
		Robot.Outputs.MotionCommand.MoveSubIndex005 := Output_Params[5];
		Robot.Outputs.MotionCommand.MoveSubIndex006 := Output_Params[6];
	    
	    IF ExternalStateControl THEN
	        IF ExternalMoveID <> 0 AND ExternalMoveID <> 32150 AND ExternalMoveID <> 32151 THEN
	            Robot.Outputs.MotionControl.MoveID := ExternalMoveID;
	            Sent := TRUE;
	        END_IF;
	        
	    ELSE (*Not External Control*)
	        IF Robot.Outputs.MotionControl.MoveID = 32150 THEN
	            Robot.Outputs.MotionControl.MoveID := 32151;
	        ELSIF Robot.Outputs.MotionControl.MoveID = 32151 THEN
	            Robot.Outputs.MotionControl.MoveID := 32150;
	        ELSIF Robot.Outputs.MotionControl.MoveID <> 32150 OR Robot.Outputs.MotionControl.MoveID <> 32151 THEN
	            Robot.Outputs.MotionControl.MoveID := 32150;
	        END_IF;
	        Sent := TRUE;
	    END_IF;
	END_IF;

	(* Check if command has been sent, if so, check if it was received *)
	IF Sent AND
	    Robot.Outputs.MotionCommand.MoveCommand = EnumToNum(Meca500Cmd#SetConf) AND
	    Robot.Outputs.MotionCommand.MoveSubIndex001 = Output_Params[1] AND 
		Robot.Outputs.MotionCommand.MoveSubIndex002 = Output_Params[2] AND 
		Robot.Outputs.MotionCommand.MoveSubIndex003 = Output_Params[3] AND 
		Robot.Outputs.MotionCommand.MoveSubIndex004 = Output_Params[4] AND 
		Robot.Outputs.MotionCommand.MoveSubIndex005 = Output_Params[5] AND 
		Robot.Outputs.MotionCommand.MoveSubIndex006 = Output_Params[6] AND
		Robot.Inputs.Motion.MoveID = Robot.Outputs.MotionControl.MoveID 
	THEN
		 Buffered := TRUE;
	END_IF;


	(*If External _Move ID is equal to Internal, raise an error*)
	IF ExternalMoveID = 32150 OR ExternalMoveID = 32151 THEN
	    Error := TRUE;
	END_IF;

	FirstScan := TRUE;
ELSE
	FirstScan := False;
	Sent := FALSE;
	Buffered := FALSE;
END_IF;
END_FUNCTION_BLOCK

FUNCTION_BLOCK Meca500_SetConfTurn
VAR
    Output_Params : array[1..6] of real;
    FirstScan : BOOL := False;
END_VAR
VAR_INPUT
    Execute : BOOL;
    Config : REAL;
END_VAR
VAR_OUTPUT
    Sent : BOOL;
    Buffered : BOOL;
    Error : BOOL;
END_VAR
VAR_IN_OUT
    Robot : Meca500;
END_VAR
VAR_INPUT
    ExternalStateControl : BOOL;
    ExternalMoveID : UINT;
END_VAR
IF Execute THEN	
	(*Collect Inputs and store them locally*)
	Output_Params[1]:=Config;
	Output_Params[2]:=0;
	Output_Params[3]:=0;
	Output_Params[4]:=0;
	Output_Params[5]:=0;
	Output_Params[6]:=0;

	(* If Values have change, Reinitialise Outputs*)

	IF FirstScan=0 OR 
		Robot.Outputs.MotionCommand.MoveSubIndex001 <> Output_Params[1] OR 
		Robot.Outputs.MotionCommand.MoveSubIndex002 <> Output_Params[2] OR 
		Robot.Outputs.MotionCommand.MoveSubIndex003 <> Output_Params[3] OR
		Robot.Outputs.MotionCommand.MoveSubIndex004 <> Output_Params[4] OR 
		Robot.Outputs.MotionCommand.MoveSubIndex005 <> Output_Params[5] OR 
		Robot.Outputs.MotionCommand.MoveSubIndex006 <> Output_Params[6] 
	THEN
		Buffered := FALSE;
		Sent := FALSE;
	END_IF;


	(*if not in legacy mode, Act Setpoint*)
	IF Robot.Outputs.MotionControl.MoveID <> 0 THEN
	    Robot.Outputs.MotionControl.SetPoint := TRUE;
	END_IF;

	(* To send _Move, send _Move ID *)
	IF NOT Buffered AND NOT Sent THEN
	    
	    Robot.Outputs.MotionCommand.MoveCommand	:= EnumToNum(Meca500Cmd#SetConfTurn);
	    Robot.Outputs.MotionCommand.MoveSubIndex001 := Output_Params[1];
		Robot.Outputs.MotionCommand.MoveSubIndex002 := Output_Params[2];
		Robot.Outputs.MotionCommand.MoveSubIndex003 := Output_Params[3];
		Robot.Outputs.MotionCommand.MoveSubIndex004 := Output_Params[4];
		Robot.Outputs.MotionCommand.MoveSubIndex005 := Output_Params[5];
		Robot.Outputs.MotionCommand.MoveSubIndex006 := Output_Params[6];
	    
	    IF ExternalStateControl THEN
	        IF ExternalMoveID <> 0 AND ExternalMoveID <> 32250 AND ExternalMoveID <> 32251 THEN
	            Robot.Outputs.MotionControl.MoveID := ExternalMoveID;
	            Sent := TRUE;
	        END_IF;
	        
	    ELSE (*Not External Control*)
	        IF Robot.Outputs.MotionControl.MoveID = 32250 THEN
	            Robot.Outputs.MotionControl.MoveID := 32251;
	        ELSIF Robot.Outputs.MotionControl.MoveID = 32251 THEN
	            Robot.Outputs.MotionControl.MoveID := 32250;
	        ELSIF Robot.Outputs.MotionControl.MoveID <> 32250 OR Robot.Outputs.MotionControl.MoveID <> 32251 THEN
	            Robot.Outputs.MotionControl.MoveID := 32250;
	        END_IF;
	        Sent := TRUE;
	    END_IF;
	END_IF;

	(* Check if command has been sent, if so, check if it was received *)
	IF Sent AND
	    Robot.Outputs.MotionCommand.MoveCommand = EnumToNum(Meca500Cmd#SetConfTurn) AND
	    Robot.Outputs.MotionCommand.MoveSubIndex001 = Output_Params[1] AND 
		Robot.Outputs.MotionCommand.MoveSubIndex002 = Output_Params[2] AND 
		Robot.Outputs.MotionCommand.MoveSubIndex003 = Output_Params[3] AND 
		Robot.Outputs.MotionCommand.MoveSubIndex004 = Output_Params[4] AND 
		Robot.Outputs.MotionCommand.MoveSubIndex005 = Output_Params[5] AND 
		Robot.Outputs.MotionCommand.MoveSubIndex006 = Output_Params[6] AND
		Robot.Inputs.Motion.MoveID = Robot.Outputs.MotionControl.MoveID 
	THEN
		 Buffered := TRUE;
	END_IF;


	(*If External _Move ID is equal to Internal, raise an error*)
	IF ExternalMoveID = 32250 OR ExternalMoveID = 32251 THEN
	    Error := TRUE;
	END_IF;

	FirstScan := TRUE;
ELSE
	FirstScan := False;
	Sent := FALSE;
	Buffered := FALSE;
END_IF;
END_FUNCTION_BLOCK

FUNCTION_BLOCK Meca500_SetGripperForce
VAR
    Output_Params : array[1..6] of real;
    FirstScan : BOOL := False;
END_VAR
VAR_INPUT
    Execute : BOOL;
    Force : REAL;
END_VAR
VAR_OUTPUT
    Sent : BOOL;
    Buffered : BOOL;
    Error : BOOL;
END_VAR
VAR_IN_OUT
    Robot : Meca500;
END_VAR
VAR_INPUT
    ExternalStateControl : BOOL;
    ExternalMoveID : UINT;
END_VAR
IF Execute THEN	
	(*Collect Inputs and store them locally*)
	Output_Params[1]:=Force;
	Output_Params[2]:=0;
	Output_Params[3]:=0;
	Output_Params[4]:=0;
	Output_Params[5]:=0;
	Output_Params[6]:=0;

	(* If Values have change, Reinitialise Outputs*)

	IF FirstScan=0 OR 
		Robot.Outputs.MotionCommand.MoveSubIndex001 <> Output_Params[1] OR 
		Robot.Outputs.MotionCommand.MoveSubIndex002 <> Output_Params[2] OR 
		Robot.Outputs.MotionCommand.MoveSubIndex003 <> Output_Params[3] OR
		Robot.Outputs.MotionCommand.MoveSubIndex004 <> Output_Params[4] OR 
		Robot.Outputs.MotionCommand.MoveSubIndex005 <> Output_Params[5] OR 
		Robot.Outputs.MotionCommand.MoveSubIndex006 <> Output_Params[6] 
	THEN
		Buffered := FALSE;
		Sent := FALSE;
	END_IF;


	(*if not in legacy mode, Act Setpoint*)
	IF Robot.Outputs.MotionControl.MoveID <> 0 THEN
	    Robot.Outputs.MotionControl.SetPoint := TRUE;
	END_IF;

	(* To send _Move, send _Move ID *)
	IF NOT Buffered AND NOT Sent THEN
	    
	    Robot.Outputs.MotionCommand.MoveCommand	:= EnumToNum(Meca500Cmd#SetGripperForce);
	    Robot.Outputs.MotionCommand.MoveSubIndex001 := Output_Params[1];
		Robot.Outputs.MotionCommand.MoveSubIndex002 := Output_Params[2];
		Robot.Outputs.MotionCommand.MoveSubIndex003 := Output_Params[3];
		Robot.Outputs.MotionCommand.MoveSubIndex004 := Output_Params[4];
		Robot.Outputs.MotionCommand.MoveSubIndex005 := Output_Params[5];
		Robot.Outputs.MotionCommand.MoveSubIndex006 := Output_Params[6];
	    
	    IF ExternalStateControl THEN
	        IF ExternalMoveID <> 0 AND ExternalMoveID <> 32200 AND ExternalMoveID <> 32201 THEN
	            Robot.Outputs.MotionControl.MoveID := ExternalMoveID;
	            Sent := TRUE;
	        END_IF;
	        
	    ELSE (*Not External Control*)
	        IF Robot.Outputs.MotionControl.MoveID = 32200 THEN
	            Robot.Outputs.MotionControl.MoveID := 32201;
	        ELSIF Robot.Outputs.MotionControl.MoveID = 32201 THEN
	            Robot.Outputs.MotionControl.MoveID := 32200;
	        ELSIF Robot.Outputs.MotionControl.MoveID <> 32200 OR Robot.Outputs.MotionControl.MoveID <> 32201 THEN
	            Robot.Outputs.MotionControl.MoveID := 32200;
	        END_IF;
	        Sent := TRUE;
	    END_IF;
	END_IF;

	(* Check if command has been sent, if so, check if it was received *)
	IF Sent AND
	    Robot.Outputs.MotionCommand.MoveCommand = EnumToNum(Meca500Cmd#SetGripperForce) AND
	    Robot.Outputs.MotionCommand.MoveSubIndex001 = Output_Params[1] AND 
		Robot.Outputs.MotionCommand.MoveSubIndex002 = Output_Params[2] AND 
		Robot.Outputs.MotionCommand.MoveSubIndex003 = Output_Params[3] AND 
		Robot.Outputs.MotionCommand.MoveSubIndex004 = Output_Params[4] AND 
		Robot.Outputs.MotionCommand.MoveSubIndex005 = Output_Params[5] AND 
		Robot.Outputs.MotionCommand.MoveSubIndex006 = Output_Params[6] AND
		Robot.Inputs.Motion.MoveID = Robot.Outputs.MotionControl.MoveID 
	THEN
		 Buffered := TRUE;
	END_IF;


	(*If External _Move ID is equal to Internal, raise an error*)
	IF ExternalMoveID = 32200 OR ExternalMoveID = 32201 THEN
	    Error := TRUE;
	END_IF;

	FirstScan := TRUE;
ELSE
	FirstScan := False;
	Sent := FALSE;
	Buffered := FALSE;
END_IF;
END_FUNCTION_BLOCK

FUNCTION_BLOCK Meca500_SetGripperRange
VAR
    Output_Params : array[1..6] of real;
    FirstScan : BOOL := False;
END_VAR
VAR_INPUT
    Execute : BOOL;
    Minimum : REAL;
    Maximum : REAL;
END_VAR
VAR_OUTPUT
    Sent : BOOL;
    Buffered : BOOL;
    Error : BOOL;
END_VAR
VAR_IN_OUT
    Robot : Meca500;
END_VAR
VAR_INPUT
    ExternalStateControl : BOOL;
    ExternalMoveID : UINT;
END_VAR
IF Execute THEN	
	(*Collect Inputs and store them locally*)
	Output_Params[1]:=Minimum;
	Output_Params[2]:=Maximum;
	Output_Params[3]:=0;
	Output_Params[4]:=0;
	Output_Params[5]:=0;
	Output_Params[6]:=0;

	(* If Values have change, Reinitialise Outputs*)

	IF FirstScan=0 OR 
		Robot.Outputs.MotionCommand.MoveSubIndex001 <> Output_Params[1] OR 
		Robot.Outputs.MotionCommand.MoveSubIndex002 <> Output_Params[2] OR 
		Robot.Outputs.MotionCommand.MoveSubIndex003 <> Output_Params[3] OR
		Robot.Outputs.MotionCommand.MoveSubIndex004 <> Output_Params[4] OR 
		Robot.Outputs.MotionCommand.MoveSubIndex005 <> Output_Params[5] OR 
		Robot.Outputs.MotionCommand.MoveSubIndex006 <> Output_Params[6] 
	THEN
		Buffered := FALSE;
		Sent := FALSE;
	END_IF;


	(*if not in legacy mode, Act Setpoint*)
	IF Robot.Outputs.MotionControl.MoveID <> 0 THEN
	    Robot.Outputs.MotionControl.SetPoint := TRUE;
	END_IF;

	(* To send _Move, send _Move ID *)
	IF NOT Buffered AND NOT Sent THEN
	    
